LIN {X 0,Y 573.237,Z 371.706,A -85,B 0,C 180,E1 -2343.515,E2 -2343.515} C_VEL
LIN {X 0,Y 573.293,Z 371.696,A -85,B 0,C 180,E1 -2345.628,E2 -2345.628} C_VEL
LIN {X 0,Y 573.287,Z 371.699,A -85,B 0,C 180,E1 -2348.46,E2 -2348.46} C_VEL
LIN {X 0,Y 573.275,Z 371.704,A -85,B 0,C 180,E1 -2351.312,E2 -2351.312} C_VEL
LIN {X 0,Y 573.284,Z 371.701,A -85,B 0,C 180,E1 -2354.424,E2 -2354.424} C_VEL
LIN {X 0,Y 573.262,Z 371.699,A -85,B 0,C 180,E1 -2357.112,E2 -2357.112} C_VEL
LIN {X 0,Y 573.254,Z 371.701,A -85,B 0,C 180,E1 -2360.077,E2 -2360.077} C_VEL
LIN {X 0,Y 573.237,Z 371.705,A -85,B 0,C 180,E1 -2363.099,E2 -2363.099} C_VEL
LIN {X 0,Y 573.254,Z 371.702,A -85,B 0,C 180,E1 -2364.391,E2 -2364.391} C_VEL
LIN {X 0,Y 572.627,Z 371.783,A -85,B 0,C 180,E1 -2364.977,E2 -2364.977} C_VEL
LIN {X 0,Y 569.784,Z 372.141,A -85,B 0,C 180,E1 -2365.928,E2 -2365.928} C_VEL
LIN {X 0,Y 567.352,Z 372.443,A -85,B 0,C 180,E1 -2366.694,E2 -2366.694} C_VEL
LIN {X 0,Y 566.296,Z 372.571,A -85,B 0,C 180,E1 -2367.285,E2 -2367.285} C_VEL
LIN {X 0,Y 566.206,Z 372.581,A -85,B 0,C 180,E1 -2367.485,E2 -2367.485} C_VEL
LIN {X 0,Y 566.203,Z 372.58,A -85,B 0,C 180,E1 -2369.769,E2 -2369.769} C_VEL
LIN {X 0,Y 566.207,Z 372.585,A -85,B 0,C 180,E1 -2372.43,E2 -2372.43} C_VEL
LIN {X 0,Y 566.216,Z 372.578,A -85,B 0,C 180,E1 -2374.994,E2 -2374.994} C_VEL
LIN {X 0,Y 566.199,Z 372.584,A -85,B 0,C 180,E1 -2377.461,E2 -2377.461} C_VEL
LIN {X 0,Y 566.22,Z 372.579,A -85,B 0,C 180,E1 -2380.198,E2 -2380.198} C_VEL
LIN {X 0,Y 566.204,Z 372.579,A -85,B 0,C 180,E1 -2383.054,E2 -2383.054} C_VEL
LIN {X 0,Y 566.205,Z 372.58,A -85,B 0,C 180,E1 -2386.048,E2 -2386.048} C_VEL
LIN {X 0,Y 566.214,Z 372.583,A -85,B 0,C 180,E1 -2388.864,E2 -2388.864} C_VEL
LIN {X 0,Y 566.217,Z 372.582,A -85,B 0,C 180,E1 -2390.726,E2 -2390.726} C_VEL
LIN {X 0,Y 566.225,Z 373.259,A -85,B 0,C 180,E1 -2391.64,E2 -2391.64} C_VEL
LIN {X 0,Y 566.24,Z 377.975,A -85,B 0,C 180,E1 -2394.313,E2 -2394.313} C_VEL
LIN {X 0,Y 566.231,Z 382.684,A -85,B 0,C 180,E1 -2396.899,E2 -2396.899} C_VEL
LIN {X 0,Y 566.13,Z 387.389,A -85,B 0,C 180,E1 -2399.404,E2 -2399.404} C_VEL
LIN {X 0,Y 566.119,Z 392.066,A -85,B 0,C 180,E1 -2401.852,E2 -2401.852} C_VEL
LIN {X 0,Y 566.079,Z 398.311,A -85,B 0,C 180,E1 -2405.032,E2 -2405.032} C_VEL
LIN {X 0,Y 566.009,Z 403.027,A -85,B 0,C 180,E1 -2407.361,E2 -2407.361} C_VEL
LIN {X 0,Y 565.977,Z 407.753,A -85,B 0,C 180,E1 -2409.654,E2 -2409.654} C_VEL
LIN {X 0,Y 565.975,Z 412.48,A -85,B 0,C 180,E1 -2411.914,E2 -2411.914} C_VEL
LIN {X 0,Y 565.96,Z 418.537,A -85,B 0,C 180,E1 -2414.769,E2 -2414.769} C_VEL
LIN {X 0,Y 567.389,Z 426.398,A -85,B 0,C 180,E1 -2414.95,E2 -2414.95} C_VEL
LIN {X 0,Y 567.256,Z 440.824,A -85,B 0,C 180,E1 -2415.314,E2 -2415.314} C_VEL
LIN {X 0,Y 567.092,Z 455.098,A -85,B 0,C 180,E1 -2415.832,E2 -2415.832} C_VEL
LIN {X 0,Y 566.914,Z 468.271,A -85,B 0,C 180,E1 -2416.468,E2 -2416.468} C_VEL
LIN {X 0,Y 566.715,Z 480.213,A -85,B 0,C 180,E1 -2417.193,E2 -2417.193} C_VEL
LIN {X 0,Y 566.536,Z 492.291,A -85,B 0,C 180,E1 -2418.098,E2 -2418.098} C_VEL
LIN {X 0,Y 566.399,Z 503.503,A -85,B 0,C 180,E1 -2419.126,E2 -2419.126} C_VEL
LIN {X 0,Y 566.202,Z 512.969,A -85,B 0,C 180,E1 -2420.173,E2 -2420.173} C_VEL
LIN {X 0,Y 566.123,Z 521.1,A -85,B 0,C 180,E1 -2421.253,E2 -2421.253} C_VEL
LIN {X 0,Y 566.016,Z 528.883,A -85,B 0,C 180,E1 -2422.509,E2 -2422.509} C_VEL
LIN {X 0,Y 565.945,Z 534.324,A -85,B 0,C 180,E1 -2423.583,E2 -2423.583} C_VEL
LIN {X 0,Y 565.928,Z 538.8,A -85,B 0,C 180,E1 -2424.656,E2 -2424.656} C_VEL
LIN {X 0,Y 565.957,Z 542.311,A -85,B 0,C 180,E1 -2425.727,E2 -2425.727} C_VEL
LIN {X 0,Y 565.875,Z 545.743,A -85,B 0,C 180,E1 -2427.153,E2 -2427.153} C_VEL
LIN {X 0,Y 565.844,Z 547.784,A -85,B 0,C 180,E1 -2428.577,E2 -2428.577} C_VEL
LIN {X 0,Y 565.838,Z 548.496,A -85,B 0,C 180,E1 -2430,E2 -2430} C_VEL
LIN {X 0,Y 565.841,Z 547.88,A -85,B 0,C 180,E1 -2431.423,E2 -2431.423} C_VEL
LIN {X 0,Y 565.873,Z 545.922,A -85,B 0,C 180,E1 -2432.848,E2 -2432.848} C_VEL
LIN {X 0,Y 565.958,Z 542.576,A -85,B 0,C 180,E1 -2434.273,E2 -2434.273} C_VEL
LIN {X 0,Y 565.984,Z 537.747,A -85,B 0,C 180,E1 -2435.701,E2 -2435.701} C_VEL
LIN {X 0,Y 565.981,Z 531.28,A -85,B 0,C 180,E1 -2437.133,E2 -2437.133} C_VEL
LIN {X 0,Y 566.093,Z 524.08,A -85,B 0,C 180,E1 -2438.388,E2 -2438.388} C_VEL
LIN {X 0,Y 566.172,Z 516.54,A -85,B 0,C 180,E1 -2439.467,E2 -2439.467} C_VEL
LIN {X 0,Y 566.29,Z 507.484,A -85,B 0,C 180,E1 -2440.548,E2 -2440.548} C_VEL
LIN {X 0,Y 566.486,Z 498.473,A -85,B 0,C 180,E1 -2441.449,E2 -2441.449} C_VEL
LIN {X 0,Y 566.626,Z 487.721,A -85,B 0,C 180,E1 -2442.354,E2 -2442.354} C_VEL
LIN {X 0,Y 566.767,Z 475.957,A -85,B 0,C 180,E1 -2443.171,E2 -2443.171} C_VEL
LIN {X 0,Y 566.999,Z 462.98,A -85,B 0,C 180,E1 -2443.896,E2 -2443.896} C_VEL
LIN {X 0,Y 567.199,Z 450.296,A -85,B 0,C 180,E1 -2444.451,E2 -2444.451} C_VEL
LIN {X 0,Y 567.312,Z 436.696,A -85,B 0,C 180,E1 -2444.899,E2 -2444.899} C_VEL
LIN {X 0,Y 567.239,Z 424.971,A -85,B 0,C 180,E1 -2445.173,E2 -2445.173} C_VEL
LIN {X 0,Y 565.933,Z 418.532,A -85,B 0,C 180,E1 -2445.324,E2 -2445.324} C_VEL
LIN {X 0,Y 565.976,Z 412.669,A -85,B 0,C 180,E1 -2448.086,E2 -2448.086} C_VEL
LIN {X 0,Y 566.015,Z 406.364,A -85,B 0,C 180,E1 -2451.105,E2 -2451.105} C_VEL
LIN {X 0,Y 566.038,Z 400.057,A -85,B 0,C 180,E1 -2454.188,E2 -2454.188} C_VEL
LIN {X 0,Y 566.072,Z 395.207,A -85,B 0,C 180,E1 -2456.631,E2 -2456.631} C_VEL
LIN {X 0,Y 566.118,Z 390.688,A -85,B 0,C 180,E1 -2458.958,E2 -2458.958} C_VEL
LIN {X 0,Y 566.157,Z 385.986,A -85,B 0,C 180,E1 -2461.424,E2 -2461.424} C_VEL
LIN {X 0,Y 566.216,Z 381.278,A -85,B 0,C 180,E1 -2463.956,E2 -2463.956} C_VEL
LIN {X 0,Y 566.252,Z 376.566,A -85,B 0,C 180,E1 -2466.566,E2 -2466.566} C_VEL
LIN {X 0,Y 566.218,Z 373.075,A -85,B 0,C 180,E1 -2468.559,E2 -2468.559} C_VEL
LIN {X 0,Y 566.222,Z 372.584,A -85,B 0,C 180,E1 -2469.686,E2 -2469.686} C_VEL
LIN {X 0,Y 566.209,Z 372.584,A -85,B 0,C 180,E1 -2472.918,E2 -2472.918} C_VEL
LIN {X 0,Y 566.198,Z 372.584,A -85,B 0,C 180,E1 -2476.049,E2 -2476.049} C_VEL
LIN {X 0,Y 566.182,Z 372.583,A -85,B 0,C 180,E1 -2478.861,E2 -2478.861} C_VEL
LIN {X 0,Y 566.189,Z 372.582,A -85,B 0,C 180,E1 -2481.637,E2 -2481.637} C_VEL
LIN {X 0,Y 566.216,Z 372.583,A -85,B 0,C 180,E1 -2484.312,E2 -2484.312} C_VEL
LIN {X 0,Y 566.224,Z 372.577,A -85,B 0,C 180,E1 -2486.898,E2 -2486.898} C_VEL
LIN {X 0,Y 566.185,Z 372.586,A -85,B 0,C 180,E1 -2489.407,E2 -2489.407} C_VEL
LIN {X 0,Y 566.215,Z 372.578,A -85,B 0,C 180,E1 -2491.857,E2 -2491.857} C_VEL
LIN {X 0,Y 566.218,Z 372.582,A -85,B 0,C 180,E1 -2494.251,E2 -2494.251} C_VEL
LIN {X 0,Y 566.177,Z 372.582,A -85,B 0,C 180,E1 -2496.718,E2 -2496.718} C_VEL
LIN {X 0,Y 566.216,Z 372.577,A -85,B 0,C 180,E1 -2499.663,E2 -2499.663} C_VEL
LIN {X 0,Y 566.203,Z 372.58,A -85,B 0,C 180,E1 -2502.668,E2 -2502.668} C_VEL
LIN {X 0,Y 566.238,Z 372.579,A -85,B 0,C 180,E1 -2505.627,E2 -2505.627} C_VEL
LIN {X 0,Y 566.239,Z 372.581,A -85,B 0,C 180,E1 -2508.675,E2 -2508.675} C_VEL
LIN {X 0,Y 566.231,Z 372.576,A -85,B 0,C 180,E1 -2511.434,E2 -2511.434} C_VEL
LIN {X 0,Y 566.261,Z 372.572,A -85,B 0,C 180,E1 -2514.302,E2 -2514.302} C_VEL
LIN {X 0,Y 566.279,Z 372.57,A -85,B 0,C 180,E1 -2517.866,E2 -2517.866} C_VEL
LIN {X 0,Y 566.305,Z 372.566,A -85,B 0,C 180,E1 -2520.711,E2 -2520.711} C_VEL
LIN {X 0,Y 566.278,Z 372.571,A -85,B 0,C 180,E1 -2522.845,E2 -2522.845} C_VEL
LIN {X 0,Y 566.26,Z 372.572,A -85,B 0,C 180,E1 -2525.698,E2 -2525.698} C_VEL
LIN {X 0,Y 566.21,Z 372.58,A -85,B 0,C 180,E1 -2528.566,E2 -2528.566} C_VEL
LIN {X 0,Y 566.246,Z 372.579,A -85,B 0,C 180,E1 -2531.454,E2 -2531.454} C_VEL
LIN {X 0,Y 566.238,Z 372.58,A -85,B 0,C 180,E1 -2534.506,E2 -2534.506} C_VEL
LIN {X 0,Y 566.207,Z 372.579,A -85,B 0,C 180,E1 -2537.331,E2 -2537.331} C_VEL
LIN {X 0,Y 566.217,Z 372.577,A -85,B 0,C 180,E1 -2540.337,E2 -2540.337} C_VEL
LIN {X 0,Y 566.193,Z 372.58,A -85,B 0,C 180,E1 -2543.404,E2 -2543.404} C_VEL
LIN {X 0,Y 566.212,Z 372.582,A -85,B 0,C 180,E1 -2545.749,E2 -2545.749} C_VEL
LIN {X 0,Y 566.206,Z 372.579,A -85,B 0,C 180,E1 -2548.202,E2 -2548.202} C_VEL
LIN {X 0,Y 566.195,Z 372.584,A -85,B 0,C 180,E1 -2551.076,E2 -2551.076} C_VEL
LIN {X 0,Y 566.215,Z 372.58,A -85,B 0,C 180,E1 -2553.734,E2 -2553.734} C_VEL
LIN {X 0,Y 566.219,Z 372.578,A -85,B 0,C 180,E1 -2556.568,E2 -2556.568} C_VEL
LIN {X 0,Y 566.216,Z 372.578,A -85,B 0,C 180,E1 -2559.686,E2 -2559.686} C_VEL
LIN {X 0,Y 566.213,Z 372.584,A -85,B 0,C 180,E1 -2562.087,E2 -2562.087} C_VEL
LIN {X 0,Y 566.171,Z 372.585,A -85,B 0,C 180,E1 -2565.036,E2 -2565.036} C_VEL
LIN {X 0,Y 566.221,Z 372.579,A -85,B 0,C 180,E1 -2568.136,E2 -2568.136} C_VEL
LIN {X 0,Y 566.243,Z 372.603,A -85,B 0,C 180,E1 -2570.822,E2 -2570.822} C_VEL
LIN {X 0,Y 566.383,Z 376.17,A -85,B 0,C 180,E1 -2572.575,E2 -2572.575} C_VEL
LIN {X 0,Y 566.341,Z 381.706,A -85,B 0,C 180,E1 -2575.191,E2 -2575.191} C_VEL
LIN {X 0,Y 566.263,Z 387.274,A -85,B 0,C 180,E1 -2577.745,E2 -2577.745} C_VEL
LIN {X 0,Y 566.206,Z 393.116,A -85,B 0,C 180,E1 -2580.328,E2 -2580.328} C_VEL
LIN {X 0,Y 566.15,Z 400.382,A -85,B 0,C 180,E1 -2583.455,E2 -2583.455} C_VEL
LIN {X 0,Y 566.105,Z 405.984,A -85,B 0,C 180,E1 -2585.815,E2 -2585.815} C_VEL
LIN {X 0,Y 566.077,Z 413.413,A -85,B 0,C 180,E1 -2588.897,E2 -2588.897} C_VEL
LIN {X 0,Y 566.008,Z 420.842,A -85,B 0,C 180,E1 -2591.915,E2 -2591.915} C_VEL
LIN {X 0,Y 565.956,Z 427.806,A -85,B 0,C 180,E1 -2594.699,E2 -2594.699} C_VEL
LIN {X 0,Y 567.417,Z 435.018,A -85,B 0,C 180,E1 -2594.878,E2 -2594.878} C_VEL
LIN {X 0,Y 567.262,Z 449.476,A -85,B 0,C 180,E1 -2595.228,E2 -2595.228} C_VEL
LIN {X 0,Y 567.086,Z 463.96,A -85,B 0,C 180,E1 -2595.74,E2 -2595.74} C_VEL
LIN {X 0,Y 566.927,Z 477.39,A -85,B 0,C 180,E1 -2596.377,E2 -2596.377} C_VEL
LIN {X 0,Y 566.741,Z 489.51,A -85,B 0,C 180,E1 -2597.102,E2 -2597.102} C_VEL
LIN {X 0,Y 566.541,Z 501.751,A -85,B 0,C 180,E1 -2598.007,E2 -2598.007} C_VEL
LIN {X 0,Y 566.433,Z 512.501,A -85,B 0,C 180,E1 -2598.98,E2 -2598.98} C_VEL
LIN {X 0,Y 566.206,Z 521.851,A -85,B 0,C 180,E1 -2599.993,E2 -2599.993} C_VEL
LIN {X 0,Y 566.137,Z 530.172,A -85,B 0,C 180,E1 -2601.073,E2 -2601.073} C_VEL
LIN {X 0,Y 566.046,Z 538.126,A -85,B 0,C 180,E1 -2602.33,E2 -2602.33} C_VEL
LIN {X 0,Y 565.944,Z 544.527,A -85,B 0,C 180,E1 -2603.583,E2 -2603.583} C_VEL
LIN {X 0,Y 565.928,Z 548.961,A -85,B 0,C 180,E1 -2604.656,E2 -2604.656} C_VEL
LIN {X 0,Y 565.956,Z 552.443,A -85,B 0,C 180,E1 -2605.727,E2 -2605.727} C_VEL
LIN {X 0,Y 565.875,Z 555.832,A -85,B 0,C 180,E1 -2607.152,E2 -2607.152} C_VEL
LIN {X 0,Y 565.841,Z 557.833,A -85,B 0,C 180,E1 -2608.576,E2 -2608.576} C_VEL
LIN {X 0,Y 565.837,Z 558.5,A -85,B 0,C 180,E1 -2610,E2 -2610} C_VEL
LIN {X 0,Y 565.841,Z 557.833,A -85,B 0,C 180,E1 -2611.423,E2 -2611.423} C_VEL
LIN {X 0,Y 565.875,Z 555.834,A -85,B 0,C 180,E1 -2612.847,E2 -2612.847} C_VEL
LIN {X 0,Y 565.956,Z 552.445,A -85,B 0,C 180,E1 -2614.273,E2 -2614.273} C_VEL
LIN {X 0,Y 565.985,Z 547.568,A -85,B 0,C 180,E1 -2615.701,E2 -2615.701} C_VEL
LIN {X 0,Y 565.995,Z 543.045,A -85,B 0,C 180,E1 -2616.739,E2 -2616.739} C_VEL
LIN {X 0,Y 566.047,Z 536.037,A -85,B 0,C 180,E1 -2618.029,E2 -2618.029} C_VEL
LIN {X 0,Y 566.177,Z 527.559,A -85,B 0,C 180,E1 -2619.286,E2 -2619.286} C_VEL
LIN {X 0,Y 566.294,Z 518.708,A -85,B 0,C 180,E1 -2620.367,E2 -2620.367} C_VEL
LIN {X 0,Y 566.485,Z 507.99,A -85,B 0,C 180,E1 -2621.449,E2 -2621.449} C_VEL
LIN {X 0,Y 566.626,Z 497.142,A -85,B 0,C 180,E1 -2622.354,E2 -2622.354} C_VEL
LIN {X 0,Y 566.773,Z 485.258,A -85,B 0,C 180,E1 -2623.171,E2 -2623.171} C_VEL
LIN {X 0,Y 567.047,Z 472.096,A -85,B 0,C 180,E1 -2623.894,E2 -2623.894} C_VEL
LIN {X 0,Y 567.174,Z 459.298,A -85,B 0,C 180,E1 -2624.445,E2 -2624.445} C_VEL
LIN {X 0,Y 567.347,Z 445.435,A -85,B 0,C 180,E1 -2624.886,E2 -2624.886} C_VEL
LIN {X 0,Y 567.246,Z 434.169,A -85,B 0,C 180,E1 -2625.144,E2 -2625.144} C_VEL
LIN {X 0,Y 565.957,Z 427.806,A -85,B 0,C 180,E1 -2625.3,E2 -2625.3} C_VEL
LIN {X 0,Y 566.008,Z 420.842,A -85,B 0,C 180,E1 -2628.084,E2 -2628.084} C_VEL
LIN {X 0,Y 566.077,Z 413.413,A -85,B 0,C 180,E1 -2631.103,E2 -2631.103} C_VEL
LIN {X 0,Y 566.107,Z 405.985,A -85,B 0,C 180,E1 -2634.185,E2 -2634.185} C_VEL
LIN {X 0,Y 566.144,Z 400.137,A -85,B 0,C 180,E1 -2636.646,E2 -2636.646} C_VEL
LIN {X 0,Y 566.203,Z 392.884,A -85,B 0,C 180,E1 -2639.769,E2 -2639.769} C_VEL
LIN {X 0,Y 566.26,Z 386.865,A -85,B 0,C 180,E1 -2642.439,E2 -2642.439} C_VEL
LIN {X 0,Y 566.369,Z 381.254,A -85,B 0,C 180,E1 -2645.017,E2 -2645.017} C_VEL
LIN {X 0,Y 566.383,Z 376.125,A -85,B 0,C 180,E1 -2647.446,E2 -2647.446} C_VEL
LIN {X 0,Y 566.232,Z 372.582,A -85,B 0,C 180,E1 -2649.226,E2 -2649.226} C_VEL
LIN {X 0,Y 566.215,Z 372.579,A -85,B 0,C 180,E1 -2652.087,E2 -2652.087} C_VEL
LIN {X 0,Y 566.17,Z 372.586,A -85,B 0,C 180,E1 -2655.036,E2 -2655.036} C_VEL
LIN {X 0,Y 566.219,Z 372.58,A -85,B 0,C 180,E1 -2658.136,E2 -2658.136} C_VEL
LIN {X 0,Y 566.224,Z 372.579,A -85,B 0,C 180,E1 -2660.727,E2 -2660.727} C_VEL
LIN {X 0,Y 566.22,Z 372.578,A -85,B 0,C 180,E1 -2663.783,E2 -2663.783} C_VEL
LIN {X 0,Y 566.214,Z 372.581,A -85,B 0,C 180,E1 -2666.266,E2 -2666.266} C_VEL
LIN {X 0,Y 566.194,Z 372.584,A -85,B 0,C 180,E1 -2668.923,E2 -2668.923} C_VEL
LIN {X 0,Y 566.213,Z 372.578,A -85,B 0,C 180,E1 -2671.857,E2 -2671.857} C_VEL
LIN {X 0,Y 566.212,Z 372.582,A -85,B 0,C 180,E1 -2674.251,E2 -2674.251} C_VEL
LIN {X 0,Y 566.175,Z 372.583,A -85,B 0,C 180,E1 -2676.718,E2 -2676.718} C_VEL
LIN {X 0,Y 566.216,Z 372.577,A -85,B 0,C 180,E1 -2679.663,E2 -2679.663} C_VEL
LIN {X 0,Y 566.205,Z 372.58,A -85,B 0,C 180,E1 -2682.669,E2 -2682.669} C_VEL
LIN {X 0,Y 566.237,Z 372.578,A -85,B 0,C 180,E1 -2685.627,E2 -2685.627} C_VEL
LIN {X 0,Y 566.237,Z 372.581,A -85,B 0,C 180,E1 -2688.675,E2 -2688.675} C_VEL
LIN {X 0,Y 566.23,Z 372.577,A -85,B 0,C 180,E1 -2691.434,E2 -2691.434} C_VEL
LIN {X 0,Y 566.259,Z 372.572,A -85,B 0,C 180,E1 -2694.302,E2 -2694.302} C_VEL
LIN {X 0,Y 566.281,Z 372.57,A -85,B 0,C 180,E1 -2697.866,E2 -2697.866} C_VEL
LIN {X 0,Y 566.304,Z 372.567,A -85,B 0,C 180,E1 -2700.711,E2 -2700.711} C_VEL
LIN {X 0,Y 566.276,Z 372.571,A -85,B 0,C 180,E1 -2702.846,E2 -2702.846} C_VEL
LIN {X 0,Y 566.261,Z 372.572,A -85,B 0,C 180,E1 -2705.698,E2 -2705.698} C_VEL
LIN {X 0,Y 566.231,Z 372.577,A -85,B 0,C 180,E1 -2708.566,E2 -2708.566} C_VEL
LIN {X 0,Y 566.245,Z 372.579,A -85,B 0,C 180,E1 -2711.454,E2 -2711.454} C_VEL
LIN {X 0,Y 566.237,Z 372.579,A -85,B 0,C 180,E1 -2714.507,E2 -2714.507} C_VEL
LIN {X 0,Y 566.206,Z 372.579,A -85,B 0,C 180,E1 -2717.332,E2 -2717.332} C_VEL
LIN {X 0,Y 566.216,Z 372.577,A -85,B 0,C 180,E1 -2720.337,E2 -2720.337} C_VEL
LIN {X 0,Y 566.192,Z 372.581,A -85,B 0,C 180,E1 -2723.404,E2 -2723.404} C_VEL
LIN {X 0,Y 566.216,Z 372.581,A -85,B 0,C 180,E1 -2725.749,E2 -2725.749} C_VEL
LIN {X 0,Y 566.206,Z 372.581,A -85,B 0,C 180,E1 -2727.485,E2 -2727.485} C_VEL
LIN {X 0,Y 565.525,Z 372.665,A -85,B 0,C 180,E1 -2728.079,E2 -2728.079} C_VEL
LIN {X 0,Y 562.659,Z 373.025,A -85,B 0,C 180,E1 -2729.043,E2 -2729.043} C_VEL
LIN {X 0,Y 560.25,Z 373.322,A -85,B 0,C 180,E1 -2729.818,E2 -2729.818} C_VEL
LIN {X 0,Y 559.222,Z 373.45,A -85,B 0,C 180,E1 -2730.417,E2 -2730.417} C_VEL
LIN {X 0,Y 559.142,Z 373.459,A -85,B 0,C 180,E1 -2730.62,E2 -2730.62} C_VEL
LIN {X 0,Y 559.165,Z 373.457,A -85,B 0,C 180,E1 -2733.575,E2 -2733.575} C_VEL
LIN {X 0,Y 559.172,Z 373.455,A -85,B 0,C 180,E1 -2736.449,E2 -2736.449} C_VEL
LIN {X 0,Y 559.181,Z 373.46,A -85,B 0,C 180,E1 -2738.934,E2 -2738.934} C_VEL
LIN {X 0,Y 559.189,Z 373.454,A -85,B 0,C 180,E1 -2741.768,E2 -2741.768} C_VEL
LIN {X 0,Y 559.142,Z 373.459,A -85,B 0,C 180,E1 -2744.739,E2 -2744.739} C_VEL
LIN {X 0,Y 559.167,Z 373.46,A -85,B 0,C 180,E1 -2747.257,E2 -2747.257} C_VEL
LIN {X 0,Y 559.182,Z 373.459,A -85,B 0,C 180,E1 -2750.135,E2 -2750.135} C_VEL
LIN {X 0,Y 559.156,Z 373.505,A -85,B 0,C 180,E1 -2751.194,E2 -2751.194} C_VEL
LIN {X 0,Y 559.235,Z 378.005,A -85,B 0,C 180,E1 -2753.796,E2 -2753.796} C_VEL
LIN {X 0,Y 559.182,Z 382.713,A -85,B 0,C 180,E1 -2756.426,E2 -2756.426} C_VEL
LIN {X 0,Y 559.137,Z 387.415,A -85,B 0,C 180,E1 -2758.98,E2 -2758.98} C_VEL
LIN {X 0,Y 559.033,Z 393.668,A -85,B 0,C 180,E1 -2762.28,E2 -2762.28} C_VEL
LIN {X 0,Y 559.018,Z 398.653,A -85,B 0,C 180,E1 -2764.849,E2 -2764.849} C_VEL
LIN {X 0,Y 558.947,Z 404.604,A -85,B 0,C 180,E1 -2767.839,E2 -2767.839} C_VEL
LIN {X 0,Y 558.906,Z 410.906,A -85,B 0,C 180,E1 -2770.917,E2 -2770.917} C_VEL
LIN {X 0,Y 558.873,Z 415.633,A -85,B 0,C 180,E1 -2773.188,E2 -2773.188} C_VEL
LIN {X 0,Y 558.878,Z 418.705,A -85,B 0,C 180,E1 -2774.578,E2 -2774.578} C_VEL
LIN {X 0,Y 560.559,Z 427.228,A -85,B 0,C 180,E1 -2774.778,E2 -2774.778} C_VEL
LIN {X 0,Y 560.384,Z 441.221,A -85,B 0,C 180,E1 -2775.141,E2 -2775.141} C_VEL
LIN {X 0,Y 560.209,Z 455.114,A -85,B 0,C 180,E1 -2775.654,E2 -2775.654} C_VEL
LIN {X 0,Y 560,Z 468.282,A -85,B 0,C 180,E1 -2776.298,E2 -2776.298} C_VEL
LIN {X 0,Y 559.76,Z 480.22,A -85,B 0,C 180,E1 -2777.031,E2 -2777.031} C_VEL
LIN {X 0,Y 559.558,Z 492.296,A -85,B 0,C 180,E1 -2777.948,E2 -2777.948} C_VEL
LIN {X 0,Y 559.417,Z 502.3,A -85,B 0,C 180,E1 -2778.864,E2 -2778.864} C_VEL
LIN {X 0,Y 559.201,Z 511.486,A -85,B 0,C 180,E1 -2779.866,E2 -2779.866} C_VEL
LIN {X 0,Y 559.071,Z 519.868,A -85,B 0,C 180,E1 -2780.959,E2 -2780.959} C_VEL
LIN {X 0,Y 558.973,Z 527.878,A -85,B 0,C 180,E1 -2782.232,E2 -2782.232} C_VEL
LIN {X 0,Y 558.873,Z 534.327,A -85,B 0,C 180,E1 -2783.502,E2 -2783.502} C_VEL
LIN {X 0,Y 558.859,Z 538.802,A -85,B 0,C 180,E1 -2784.588,E2 -2784.588} C_VEL
LIN {X 0,Y 558.866,Z 542.314,A -85,B 0,C 180,E1 -2785.673,E2 -2785.673} C_VEL
LIN {X 0,Y 558.796,Z 545.745,A -85,B 0,C 180,E1 -2787.116,E2 -2787.116} C_VEL
LIN {X 0,Y 558.744,Z 547.785,A -85,B 0,C 180,E1 -2788.559,E2 -2788.559} C_VEL
LIN {X 0,Y 558.739,Z 548.496,A -85,B 0,C 180,E1 -2790,E2 -2790} C_VEL
LIN {X 0,Y 558.741,Z 547.879,A -85,B 0,C 180,E1 -2791.442,E2 -2791.442} C_VEL
LIN {X 0,Y 558.794,Z 545.921,A -85,B 0,C 180,E1 -2792.884,E2 -2792.884} C_VEL
LIN {X 0,Y 558.867,Z 542.575,A -85,B 0,C 180,E1 -2794.327,E2 -2794.327} C_VEL
LIN {X 0,Y 558.912,Z 537.745,A -85,B 0,C 180,E1 -2795.774,E2 -2795.774} C_VEL
LIN {X 0,Y 558.907,Z 531.278,A -85,B 0,C 180,E1 -2797.224,E2 -2797.224} C_VEL
LIN {X 0,Y 559.029,Z 524.077,A -85,B 0,C 180,E1 -2798.495,E2 -2798.495} C_VEL
LIN {X 0,Y 559.124,Z 516.536,A -85,B 0,C 180,E1 -2799.587,E2 -2799.587} C_VEL
LIN {X 0,Y 559.288,Z 507.479,A -85,B 0,C 180,E1 -2800.682,E2 -2800.682} C_VEL
LIN {X 0,Y 559.482,Z 496.513,A -85,B 0,C 180,E1 -2801.778,E2 -2801.778} C_VEL
LIN {X 0,Y 559.703,Z 485.335,A -85,B 0,C 180,E1 -2802.694,E2 -2802.694} C_VEL
LIN {X 0,Y 559.914,Z 472.981,A -85,B 0,C 180,E1 -2803.52,E2 -2803.52} C_VEL
LIN {X 0,Y 560.116,Z 461.093,A -85,B 0,C 180,E1 -2804.163,E2 -2804.163} C_VEL
LIN {X 0,Y 560.337,Z 448.009,A -85,B 0,C 180,E1 -2804.717,E2 -2804.717} C_VEL
LIN {X 0,Y 560.492,Z 434.312,A -85,B 0,C 180,E1 -2805.146,E2 -2805.146} C_VEL
LIN {X 0,Y 560.41,Z 425.983,A -85,B 0,C 180,E1 -2805.341,E2 -2805.341} C_VEL
LIN {X 0,Y 558.876,Z 418.53,A -85,B 0,C 180,E1 -2805.523,E2 -2805.523} C_VEL
LIN {X 0,Y 558.89,Z 412.668,A -85,B 0,C 180,E1 -2808.323,E2 -2808.323} C_VEL
LIN {X 0,Y 558.95,Z 406.138,A -85,B 0,C 180,E1 -2811.495,E2 -2811.495} C_VEL
LIN {X 0,Y 558.976,Z 400.098,A -85,B 0,C 180,E1 -2814.514,E2 -2814.514} C_VEL
LIN {X 0,Y 559.009,Z 395.403,A -85,B 0,C 180,E1 -2816.911,E2 -2816.911} C_VEL
LIN {X 0,Y 559.052,Z 390.721,A -85,B 0,C 180,E1 -2819.359,E2 -2819.359} C_VEL
LIN {X 0,Y 559.124,Z 386.012,A -85,B 0,C 180,E1 -2821.866,E2 -2821.866} C_VEL
LIN {X 0,Y 559.165,Z 381.307,A -85,B 0,C 180,E1 -2824.444,E2 -2824.444} C_VEL
LIN {X 0,Y 559.223,Z 376.593,A -85,B 0,C 180,E1 -2827.102,E2 -2827.102} C_VEL
LIN {X 0,Y 559.155,Z 373.463,A -85,B 0,C 180,E1 -2828.936,E2 -2828.936} C_VEL
LIN {X 0,Y 559.17,Z 373.458,A -85,B 0,C 180,E1 -2831.77,E2 -2831.77} C_VEL
LIN {X 0,Y 559.159,Z 373.459,A -85,B 0,C 180,E1 -2834.24,E2 -2834.24} C_VEL
LIN {X 0,Y 559.164,Z 373.457,A -85,B 0,C 180,E1 -2837.257,E2 -2837.257} C_VEL
LIN {X 0,Y 559.183,Z 373.454,A -85,B 0,C 180,E1 -2840.135,E2 -2840.135} C_VEL
LIN {X 0,Y 559.151,Z 373.462,A -85,B 0,C 180,E1 -2842.892,E2 -2842.892} C_VEL
LIN {X 0,Y 559.16,Z 373.458,A -85,B 0,C 180,E1 -2845.556,E2 -2845.556} C_VEL
LIN {X 0,Y 559.17,Z 373.456,A -85,B 0,C 180,E1 -2848.137,E2 -2848.137} C_VEL
LIN {X 0,Y 559.146,Z 373.462,A -85,B 0,C 180,E1 -2850.646,E2 -2850.646} C_VEL
LIN {X 0,Y 559.174,Z 373.455,A -85,B 0,C 180,E1 -2853.172,E2 -2853.172} C_VEL
LIN {X 0,Y 559.161,Z 373.46,A -85,B 0,C 180,E1 -2855.495,E2 -2855.495} C_VEL
LIN {X 0,Y 559.175,Z 373.457,A -85,B 0,C 180,E1 -2858.624,E2 -2858.624} C_VEL
LIN {X 0,Y 559.166,Z 373.458,A -85,B 0,C 180,E1 -2860.926,E2 -2860.926} C_VEL
LIN {X 0,Y 559.17,Z 373.46,A -85,B 0,C 180,E1 -2863.948,E2 -2863.948} C_VEL
LIN {X 0,Y 559.176,Z 373.454,A -85,B 0,C 180,E1 -2866.184,E2 -2866.184} C_VEL
LIN {X 0,Y 559.197,Z 373.453,A -85,B 0,C 180,E1 -2869.133,E2 -2869.133} C_VEL
LIN {X 0,Y 559.208,Z 373.455,A -85,B 0,C 180,E1 -2872.054,E2 -2872.054} C_VEL
LIN {X 0,Y 559.257,Z 373.448,A -85,B 0,C 180,E1 -2874.953,E2 -2874.953} C_VEL
LIN {X 0,Y 559.251,Z 373.446,A -85,B 0,C 180,E1 -2877.839,E2 -2877.839} C_VEL
LIN {X 0,Y 559.276,Z 373.442,A -85,B 0,C 180,E1 -2880.72,E2 -2880.72} C_VEL
LIN {X 0,Y 559.244,Z 373.448,A -85,B 0,C 180,E1 -2882.881,E2 -2882.881} C_VEL
LIN {X 0,Y 559.229,Z 373.447,A -85,B 0,C 180,E1 -2885.77,E2 -2885.77} C_VEL
LIN {X 0,Y 559.175,Z 373.455,A -85,B 0,C 180,E1 -2888.675,E2 -2888.675} C_VEL
LIN {X 0,Y 559.209,Z 373.454,A -85,B 0,C 180,E1 -2891.6,E2 -2891.6} C_VEL
LIN {X 0,Y 559.204,Z 373.457,A -85,B 0,C 180,E1 -2894.595,E2 -2894.595} C_VEL
LIN {X 0,Y 559.166,Z 373.458,A -85,B 0,C 180,E1 -2897.557,E2 -2897.557} C_VEL
LIN {X 0,Y 559.176,Z 373.457,A -85,B 0,C 180,E1 -2899.837,E2 -2899.837} C_VEL
LIN {X 0,Y 559.145,Z 373.459,A -85,B 0,C 180,E1 -2902.153,E2 -2902.153} C_VEL
LIN {X 0,Y 559.182,Z 373.454,A -85,B 0,C 180,E1 -2905.187,E2 -2905.187} C_VEL
LIN {X 0,Y 559.184,Z 373.458,A -85,B 0,C 180,E1 -2907.712,E2 -2907.712} C_VEL
LIN {X 0,Y 559.157,Z 373.456,A -85,B 0,C 180,E1 -2910.183,E2 -2910.183} C_VEL
LIN {X 0,Y 559.16,Z 373.46,A -85,B 0,C 180,E1 -2912.715,E2 -2912.715} C_VEL
LIN {X 0,Y 559.16,Z 373.459,A -85,B 0,C 180,E1 -2915.322,E2 -2915.322} C_VEL
LIN {X 0,Y 559.138,Z 373.46,A -85,B 0,C 180,E1 -2918.017,E2 -2918.017} C_VEL
LIN {X 0,Y 559.178,Z 373.458,A -85,B 0,C 180,E1 -2920.81,E2 -2920.81} C_VEL
LIN {X 0,Y 559.14,Z 373.465,A -85,B 0,C 180,E1 -2923.734,E2 -2923.734} C_VEL
LIN {X 0,Y 559.15,Z 373.462,A -85,B 0,C 180,E1 -2926.803,E2 -2926.803} C_VEL
LIN {X 0,Y 559.179,Z 373.457,A -85,B 0,C 180,E1 -2929.189,E2 -2929.189} C_VEL
LIN {X 0,Y 559.226,Z 373.554,A -85,B 0,C 180,E1 -2930.722,E2 -2930.722} C_VEL
LIN {X 0,Y 559.365,Z 376.774,A -85,B 0,C 180,E1 -2932.33,E2 -2932.33} C_VEL
LIN {X 0,Y 559.341,Z 381.817,A -85,B 0,C 180,E1 -2934.757,E2 -2934.757} C_VEL
LIN {X 0,Y 559.238,Z 387.389,A -85,B 0,C 180,E1 -2937.352,E2 -2937.352} C_VEL
LIN {X 0,Y 559.173,Z 393.578,A -85,B 0,C 180,E1 -2940.138,E2 -2940.138} C_VEL
LIN {X 0,Y 559.1,Z 400.56,A -85,B 0,C 180,E1 -2943.187,E2 -2943.187} C_VEL
LIN {X 0,Y 559.013,Z 407.827,A -85,B 0,C 180,E1 -2946.277,E2 -2946.277} C_VEL
LIN {X 0,Y 558.986,Z 415.27,A -85,B 0,C 180,E1 -2949.388,E2 -2949.388} C_VEL
LIN {X 0,Y 558.945,Z 422.699,A -85,B 0,C 180,E1 -2952.436,E2 -2952.436} C_VEL
LIN {X 0,Y 558.898,Z 427.849,A -85,B 0,C 180,E1 -2954.519,E2 -2954.519} C_VEL
LIN {X 0,Y 560.553,Z 436.545,A -85,B 0,C 180,E1 -2954.719,E2 -2954.719} C_VEL
LIN {X 0,Y 560.356,Z 450.991,A -85,B 0,C 180,E1 -2955.088,E2 -2955.088} C_VEL
LIN {X 0,Y 560.209,Z 465.083,A -85,B 0,C 180,E1 -2955.608,E2 -2955.608} C_VEL
LIN {X 0,Y 560.001,Z 477.392,A -85,B 0,C 180,E1 -2956.205,E2 -2956.205} C_VEL
LIN {X 0,Y 559.803,Z 489.512,A -85,B 0,C 180,E1 -2956.939,E2 -2956.939} C_VEL
LIN {X 0,Y 559.56,Z 501.749,A -85,B 0,C 180,E1 -2957.855,E2 -2957.855} C_VEL
LIN {X 0,Y 559.414,Z 512.773,A -85,B 0,C 180,E1 -2958.868,E2 -2958.868} C_VEL
LIN {X 0,Y 559.169,Z 523.337,A -85,B 0,C 180,E1 -2960.048,E2 -2960.048} C_VEL
LIN {X 0,Y 559.081,Z 531.407,A -85,B 0,C 180,E1 -2961.142,E2 -2961.142} C_VEL
LIN {X 0,Y 558.966,Z 539.135,A -85,B 0,C 180,E1 -2962.414,E2 -2962.414} C_VEL
LIN {X 0,Y 558.872,Z 544.527,A -85,B 0,C 180,E1 -2963.501,E2 -2963.501} C_VEL
LIN {X 0,Y 558.859,Z 548.961,A -85,B 0,C 180,E1 -2964.588,E2 -2964.588} C_VEL
LIN {X 0,Y 558.865,Z 552.443,A -85,B 0,C 180,E1 -2965.673,E2 -2965.673} C_VEL
LIN {X 0,Y 558.796,Z 555.832,A -85,B 0,C 180,E1 -2967.116,E2 -2967.116} C_VEL
LIN {X 0,Y 558.74,Z 557.833,A -85,B 0,C 180,E1 -2968.558,E2 -2968.558} C_VEL
LIN {X 0,Y 558.738,Z 558.5,A -85,B 0,C 180,E1 -2970,E2 -2970} C_VEL
LIN {X 0,Y 558.74,Z 557.834,A -85,B 0,C 180,E1 -2971.441,E2 -2971.441} C_VEL
LIN {X 0,Y 558.796,Z 555.834,A -85,B 0,C 180,E1 -2972.884,E2 -2972.884} C_VEL
LIN {X 0,Y 558.865,Z 552.445,A -85,B 0,C 180,E1 -2974.327,E2 -2974.327} C_VEL
LIN {X 0,Y 558.914,Z 547.568,A -85,B 0,C 180,E1 -2975.773,E2 -2975.773} C_VEL
LIN {X 0,Y 558.907,Z 541.054,A -85,B 0,C 180,E1 -2977.224,E2 -2977.224} C_VEL
LIN {X 0,Y 559.028,Z 533.802,A -85,B 0,C 180,E1 -2978.495,E2 -2978.495} C_VEL
LIN {X 0,Y 559.146,Z 524.823,A -85,B 0,C 180,E1 -2979.769,E2 -2979.769} C_VEL
LIN {X 0,Y 559.351,Z 515.392,A -85,B 0,C 180,E1 -2980.863,E2 -2980.863} C_VEL
LIN {X 0,Y 559.518,Z 504.952,A -85,B 0,C 180,E1 -2981.869,E2 -2981.869} C_VEL
LIN {X 0,Y 559.71,Z 493.435,A -85,B 0,C 180,E1 -2982.786,E2 -2982.786} C_VEL
LIN {X 0,Y 559.94,Z 480.643,A -85,B 0,C 180,E1 -2983.611,E2 -2983.611} C_VEL
LIN {X 0,Y 560.142,Z 468.152,A -85,B 0,C 180,E1 -2984.255,E2 -2984.255} C_VEL
LIN {X 0,Y 560.349,Z 455.044,A -85,B 0,C 180,E1 -2984.777,E2 -2984.777} C_VEL
LIN {X 0,Y 560.532,Z 440.895,A -85,B 0,C 180,E1 -2985.187,E2 -2985.187} C_VEL
LIN {X 0,Y 560.295,Z 434.755,A -85,B 0,C 180,E1 -2985.325,E2 -2985.325} C_VEL
LIN {X 0,Y 558.885,Z 427.806,A -85,B 0,C 180,E1 -2985.499,E2 -2985.499} C_VEL
LIN {X 0,Y 558.948,Z 420.842,A -85,B 0,C 180,E1 -2988.321,E2 -2988.321} C_VEL
LIN {X 0,Y 558.986,Z 415.27,A -85,B 0,C 180,E1 -2990.612,E2 -2990.612} C_VEL
LIN {X 0,Y 559.012,Z 407.811,A -85,B 0,C 180,E1 -2993.723,E2 -2993.723} C_VEL
LIN {X 0,Y 559.099,Z 400.557,A -85,B 0,C 180,E1 -2996.813,E2 -2996.813} C_VEL
LIN {X 0,Y 559.172,Z 393.57,A -85,B 0,C 180,E1 -2999.861,E2 -2999.861} C_VEL
LIN {X 0,Y 559.238,Z 387.256,A -85,B 0,C 180,E1 -3002.71,E2 -3002.71} C_VEL
LIN {X 0,Y 559.341,Z 381.68,A -85,B 0,C 180,E1 -3005.309,E2 -3005.309} C_VEL
LIN {X 0,Y 559.403,Z 376.099,A -85,B 0,C 180,E1 -3007.996,E2 -3007.996} C_VEL
LIN {X 0,Y 559.184,Z 373.46,A -85,B 0,C 180,E1 -3009.398,E2 -3009.398} C_VEL
LIN {X 0,Y 559.178,Z 373.456,A -85,B 0,C 180,E1 -3012.137,E2 -3012.137} C_VEL
LIN {X 0,Y 559.136,Z 373.461,A -85,B 0,C 180,E1 -3015.26,E2 -3015.26} C_VEL
LIN {X 0,Y 559.193,Z 373.455,A -85,B 0,C 180,E1 -3018.232,E2 -3018.232} C_VEL
LIN {X 0,Y 559.18,Z 373.459,A -85,B 0,C 180,E1 -3021.191,E2 -3021.191} C_VEL
LIN {X 0,Y 559.175,Z 373.456,A -85,B 0,C 180,E1 -3023.792,E2 -3023.792} C_VEL
LIN {X 0,Y 559.167,Z 373.457,A -85,B 0,C 180,E1 -3026.425,E2 -3026.425} C_VEL
LIN {X 0,Y 559.158,Z 373.461,A -85,B 0,C 180,E1 -3028.981,E2 -3028.981} C_VEL
LIN {X 0,Y 559.17,Z 373.455,A -85,B 0,C 180,E1 -3031.619,E2 -3031.619} C_VEL
LIN {X 0,Y 559.18,Z 373.459,A -85,B 0,C 180,E1 -3033.903,E2 -3033.903} C_VEL
LIN {X 0,Y 559.145,Z 373.458,A -85,B 0,C 180,E1 -3036.571,E2 -3036.571} C_VEL
LIN {X 0,Y 559.182,Z 373.455,A -85,B 0,C 180,E1 -3039.396,E2 -3039.396} C_VEL
LIN {X 0,Y 559.153,Z 373.458,A -85,B 0,C 180,E1 -3041.686,E2 -3041.686} C_VEL
LIN {X 0,Y 559.168,Z 373.46,A -85,B 0,C 180,E1 -3043.948,E2 -3043.948} C_VEL
LIN {X 0,Y 559.176,Z 373.454,A -85,B 0,C 180,E1 -3046.184,E2 -3046.184} C_VEL
LIN {X 0,Y 559.197,Z 373.452,A -85,B 0,C 180,E1 -3049.134,E2 -3049.134} C_VEL
LIN {X 0,Y 559.206,Z 373.454,A -85,B 0,C 180,E1 -3052.054,E2 -3052.054} C_VEL
LIN {X 0,Y 559.257,Z 373.448,A -85,B 0,C 180,E1 -3054.953,E2 -3054.953} C_VEL
LIN {X 0,Y 559.252,Z 373.445,A -85,B 0,C 180,E1 -3057.839,E2 -3057.839} C_VEL
LIN {X 0,Y 559.274,Z 373.442,A -85,B 0,C 180,E1 -3060.72,E2 -3060.72} C_VEL
LIN {X 0,Y 559.242,Z 373.448,A -85,B 0,C 180,E1 -3062.881,E2 -3062.881} C_VEL
LIN {X 0,Y 559.23,Z 373.448,A -85,B 0,C 180,E1 -3065.77,E2 -3065.77} C_VEL
LIN {X 0,Y 559.189,Z 373.453,A -85,B 0,C 180,E1 -3068.674,E2 -3068.674} C_VEL
LIN {X 0,Y 559.208,Z 373.454,A -85,B 0,C 180,E1 -3071.6,E2 -3071.6} C_VEL
LIN {X 0,Y 559.203,Z 373.457,A -85,B 0,C 180,E1 -3074.596,E2 -3074.596} C_VEL
LIN {X 0,Y 559.165,Z 373.458,A -85,B 0,C 180,E1 -3077.557,E2 -3077.557} C_VEL
LIN {X 0,Y 559.175,Z 373.457,A -85,B 0,C 180,E1 -3079.837,E2 -3079.837} C_VEL
LIN {X 0,Y 559.144,Z 373.459,A -85,B 0,C 180,E1 -3082.153,E2 -3082.153} C_VEL
LIN {X 0,Y 559.182,Z 373.454,A -85,B 0,C 180,E1 -3085.187,E2 -3085.187} C_VEL
LIN {X 0,Y 559.184,Z 373.458,A -85,B 0,C 180,E1 -3087.712,E2 -3087.712} C_VEL
LIN {X 0,Y 559.142,Z 373.459,A -85,B 0,C 180,E1 -3090.62,E2 -3090.62} C_VEL
LIN {X 0,Y 558.481,Z 373.545,A -85,B 0,C 180,E1 -3091.221,E2 -3091.221} C_VEL
LIN {X 0,Y 555.618,Z 373.901,A -85,B 0,C 180,E1 -3092.197,E2 -3092.197} C_VEL
LIN {X 0,Y 553.206,Z 374.199,A -85,B 0,C 180,E1 -3092.983,E2 -3092.983} C_VEL
LIN {X 0,Y 552.188,Z 374.326,A -85,B 0,C 180,E1 -3093.59,E2 -3093.59} C_VEL
LIN {X 0,Y 552.116,Z 374.337,A -85,B 0,C 180,E1 -3093.795,E2 -3093.795} C_VEL
LIN {X 0,Y 552.115,Z 374.335,A -85,B 0,C 180,E1 -3096.747,E2 -3096.747} C_VEL
LIN {X 0,Y 552.134,Z 374.332,A -85,B 0,C 180,E1 -3099.527,E2 -3099.527} C_VEL
LIN {X 0,Y 552.133,Z 374.336,A -85,B 0,C 180,E1 -3102.425,E2 -3102.425} C_VEL
LIN {X 0,Y 552.102,Z 374.341,A -85,B 0,C 180,E1 -3105.563,E2 -3105.563} C_VEL
LIN {X 0,Y 552.143,Z 374.337,A -85,B 0,C 180,E1 -3108.676,E2 -3108.676} C_VEL
LIN {X 0,Y 552.105,Z 374.34,A -85,B 0,C 180,E1 -3110.941,E2 -3110.941} C_VEL
LIN {X 0,Y 552.179,Z 376.458,A -85,B 0,C 180,E1 -3112.343,E2 -3112.343} C_VEL
LIN {X 0,Y 552.151,Z 381.176,A -85,B 0,C 180,E1 -3115.056,E2 -3115.056} C_VEL
LIN {X 0,Y 552.102,Z 385.883,A -85,B 0,C 180,E1 -3117.68,E2 -3117.68} C_VEL
LIN {X 0,Y 552.039,Z 390.584,A -85,B 0,C 180,E1 -3120.231,E2 -3120.231} C_VEL
LIN {X 0,Y 551.959,Z 395.875,A -85,B 0,C 180,E1 -3123.037,E2 -3123.037} C_VEL
LIN {X 0,Y 551.891,Z 401.508,A -85,B 0,C 180,E1 -3125.952,E2 -3125.952} C_VEL
LIN {X 0,Y 551.881,Z 406.294,A -85,B 0,C 180,E1 -3128.377,E2 -3128.377} C_VEL
LIN {X 0,Y 551.803,Z 412.483,A -85,B 0,C 180,E1 -3131.433,E2 -3131.433} C_VEL
LIN {X 0,Y 551.779,Z 418.392,A -85,B 0,C 180,E1 -3134.296,E2 -3134.296} C_VEL
LIN {X 0,Y 551.784,Z 418.539,A -85,B 0,C 180,E1 -3134.368,E2 -3134.368} C_VEL
LIN {X 0,Y 553.682,Z 428.899,A -85,B 0,C 180,E1 -3134.619,E2 -3134.619} C_VEL
LIN {X 0,Y 553.514,Z 442.924,A -85,B 0,C 180,E1 -3135.005,E2 -3135.005} C_VEL
LIN {X 0,Y 553.285,Z 457.197,A -85,B 0,C 180,E1 -3135.565,E2 -3135.565} C_VEL
LIN {X 0,Y 553.036,Z 469.883,A -85,B 0,C 180,E1 -3136.215,E2 -3136.215} C_VEL
LIN {X 0,Y 552.783,Z 481.521,A -85,B 0,C 180,E1 -3136.958,E2 -3136.958} C_VEL
LIN {X 0,Y 552.542,Z 493.371,A -85,B 0,C 180,E1 -3137.885,E2 -3137.885} C_VEL
LIN {X 0,Y 552.398,Z 503.77,A -85,B 0,C 180,E1 -3138.874,E2 -3138.874} C_VEL
LIN {X 0,Y 552.132,Z 512.977,A -85,B 0,C 180,E1 -3139.92,E2 -3139.92} C_VEL
LIN {X 0,Y 552.009,Z 521.107,A -85,B 0,C 180,E1 -3141.027,E2 -3141.027} C_VEL
LIN {X 0,Y 551.902,Z 528.889,A -85,B 0,C 180,E1 -3142.316,E2 -3142.316} C_VEL
LIN {X 0,Y 551.786,Z 535.436,A -85,B 0,C 180,E1 -3143.67,E2 -3143.67} C_VEL
LIN {X 0,Y 551.715,Z 540.05,A -85,B 0,C 180,E1 -3144.884,E2 -3144.884} C_VEL
LIN {X 0,Y 551.741,Z 544.21,A -85,B 0,C 180,E1 -3146.348,E2 -3146.348} C_VEL
LIN {X 0,Y 551.656,Z 546.936,A -85,B 0,C 180,E1 -3147.81,E2 -3147.81} C_VEL
LIN {X 0,Y 551.637,Z 548.306,A -85,B 0,C 180,E1 -3149.27,E2 -3149.27} C_VEL
LIN {X 0,Y 551.638,Z 548.354,A -85,B 0,C 180,E1 -3150.73,E2 -3150.73} C_VEL
LIN {X 0,Y 551.655,Z 547.069,A -85,B 0,C 180,E1 -3152.19,E2 -3152.19} C_VEL
LIN {X 0,Y 551.741,Z 544.425,A -85,B 0,C 180,E1 -3153.652,E2 -3153.652} C_VEL
LIN {X 0,Y 551.715,Z 540.352,A -85,B 0,C 180,E1 -3155.116,E2 -3155.116} C_VEL
LIN {X 0,Y 551.785,Z 535.837,A -85,B 0,C 180,E1 -3156.329,E2 -3156.329} C_VEL
LIN {X 0,Y 551.898,Z 529.381,A -85,B 0,C 180,E1 -3157.684,E2 -3157.684} C_VEL
LIN {X 0,Y 552.002,Z 521.706,A -85,B 0,C 180,E1 -3158.973,E2 -3158.973} C_VEL
LIN {X 0,Y 552.175,Z 512.213,A -85,B 0,C 180,E1 -3160.264,E2 -3160.264} C_VEL
LIN {X 0,Y 552.371,Z 501.86,A -85,B 0,C 180,E1 -3161.416,E2 -3161.416} C_VEL
LIN {X 0,Y 552.605,Z 491.19,A -85,B 0,C 180,E1 -3162.393,E2 -3162.393} C_VEL
LIN {X 0,Y 552.864,Z 478.781,A -85,B 0,C 180,E1 -3163.321,E2 -3163.321} C_VEL
LIN {X 0,Y 553.143,Z 466.484,A -85,B 0,C 180,E1 -3164.063,E2 -3164.063} C_VEL
LIN {X 0,Y 553.354,Z 452.785,A -85,B 0,C 180,E1 -3164.715,E2 -3164.715} C_VEL
LIN {X 0,Y 553.54,Z 438.632,A -85,B 0,C 180,E1 -3165.218,E2 -3165.218} C_VEL
LIN {X 0,Y 553.58,Z 427.194,A -85,B 0,C 180,E1 -3165.51,E2 -3165.51} C_VEL
LIN {X 0,Y 551.762,Z 418.529,A -85,B 0,C 180,E1 -3165.728,E2 -3165.728} C_VEL
LIN {X 0,Y 551.801,Z 414.243,A -85,B 0,C 180,E1 -3167.799,E2 -3167.799} C_VEL
LIN {X 0,Y 551.813,Z 409.514,A -85,B 0,C 180,E1 -3170.113,E2 -3170.113} C_VEL
LIN {X 0,Y 551.867,Z 404.84,A -85,B 0,C 180,E1 -3172.461,E2 -3172.461} C_VEL
LIN {X 0,Y 551.933,Z 399.258,A -85,B 0,C 180,E1 -3175.301,E2 -3175.301} C_VEL
LIN {X 0,Y 551.986,Z 393.877,A -85,B 0,C 180,E1 -3178.105,E2 -3178.105} C_VEL
LIN {X 0,Y 552.061,Z 389.182,A -85,B 0,C 180,E1 -3180.612,E2 -3180.612} C_VEL
LIN {X 0,Y 552.116,Z 384.477,A -85,B 0,C 180,E1 -3183.186,E2 -3183.186} C_VEL
LIN {X 0,Y 552.159,Z 379.763,A -85,B 0,C 180,E1 -3185.838,E2 -3185.838} C_VEL
LIN {X 0,Y 552.131,Z 375.038,A -85,B 0,C 180,E1 -3188.588,E2 -3188.588} C_VEL
LIN {X 0,Y 552.106,Z 374.341,A -85,B 0,C 180,E1 -3189.059,E2 -3189.059} C_VEL
LIN {X 0,Y 552.126,Z 374.339,A -85,B 0,C 180,E1 -3191.446,E2 -3191.446} C_VEL
LIN {X 0,Y 552.1,Z 374.342,A -85,B 0,C 180,E1 -3194.532,E2 -3194.532} C_VEL
LIN {X 0,Y 552.134,Z 374.336,A -85,B 0,C 180,E1 -3197.584,E2 -3197.584} C_VEL
LIN {X 0,Y 552.133,Z 374.332,A -85,B 0,C 180,E1 -3200.473,E2 -3200.473} C_VEL
LIN {X 0,Y 552.119,Z 374.334,A -85,B 0,C 180,E1 -3203.316,E2 -3203.316} C_VEL
LIN {X 0,Y 552.135,Z 374.337,A -85,B 0,C 180,E1 -3205.939,E2 -3205.939} C_VEL
LIN {X 0,Y 552.122,Z 374.333,A -85,B 0,C 180,E1 -3208.541,E2 -3208.541} C_VEL
LIN {X 0,Y 552.128,Z 374.333,A -85,B 0,C 180,E1 -3211.438,E2 -3211.438} C_VEL
LIN {X 0,Y 552.134,Z 374.335,A -85,B 0,C 180,E1 -3214.356,E2 -3214.356} C_VEL
LIN {X 0,Y 552.103,Z 374.335,A -85,B 0,C 180,E1 -3216.758,E2 -3216.758} C_VEL
LIN {X 0,Y 552.124,Z 374.336,A -85,B 0,C 180,E1 -3219.12,E2 -3219.12} C_VEL
LIN {X 0,Y 552.124,Z 374.333,A -85,B 0,C 180,E1 -3221.444,E2 -3221.444} C_VEL
LIN {X 0,Y 552.12,Z 374.339,A -85,B 0,C 180,E1 -3223.737,E2 -3223.737} C_VEL
LIN {X 0,Y 552.14,Z 374.331,A -85,B 0,C 180,E1 -3226.004,E2 -3226.004} C_VEL
LIN {X 0,Y 552.165,Z 374.33,A -85,B 0,C 180,E1 -3228.993,E2 -3228.993} C_VEL
LIN {X 0,Y 552.162,Z 374.335,A -85,B 0,C 180,E1 -3231.952,E2 -3231.952} C_VEL
LIN {X 0,Y 552.232,Z 374.322,A -85,B 0,C 180,E1 -3234.889,E2 -3234.889} C_VEL
LIN {X 0,Y 552.223,Z 374.321,A -85,B 0,C 180,E1 -3237.812,E2 -3237.812} C_VEL
LIN {X 0,Y 552.246,Z 374.317,A -85,B 0,C 180,E1 -3240.729,E2 -3240.729} C_VEL
LIN {X 0,Y 552.211,Z 374.324,A -85,B 0,C 180,E1 -3242.918,E2 -3242.918} C_VEL
LIN {X 0,Y 552.2,Z 374.323,A -85,B 0,C 180,E1 -3245.844,E2 -3245.844} C_VEL
LIN {X 0,Y 552.15,Z 374.33,A -85,B 0,C 180,E1 -3248.786,E2 -3248.786} C_VEL
LIN {X 0,Y 552.167,Z 374.329,A -85,B 0,C 180,E1 -3251.75,E2 -3251.75} C_VEL
LIN {X 0,Y 552.14,Z 374.336,A -85,B 0,C 180,E1 -3254.748,E2 -3254.748} C_VEL
LIN {X 0,Y 552.117,Z 374.339,A -85,B 0,C 180,E1 -3257.788,E2 -3257.788} C_VEL
LIN {X 0,Y 552.134,Z 374.332,A -85,B 0,C 180,E1 -3260.101,E2 -3260.101} C_VEL
LIN {X 0,Y 552.099,Z 374.339,A -85,B 0,C 180,E1 -3262.451,E2 -3262.451} C_VEL
LIN {X 0,Y 552.158,Z 374.329,A -85,B 0,C 180,E1 -3265.35,E2 -3265.35} C_VEL
LIN {X 0,Y 552.123,Z 374.334,A -85,B 0,C 180,E1 -3268.098,E2 -3268.098} C_VEL
LIN {X 0,Y 552.106,Z 374.338,A -85,B 0,C 180,E1 -3270.609,E2 -3270.609} C_VEL
LIN {X 0,Y 552.119,Z 374.334,A -85,B 0,C 180,E1 -3273.186,E2 -3273.186} C_VEL
LIN {X 0,Y 552.116,Z 374.339,A -85,B 0,C 180,E1 -3275.841,E2 -3275.841} C_VEL
LIN {X 0,Y 552.129,Z 374.338,A -85,B 0,C 180,E1 -3279.062,E2 -3279.062} C_VEL
LIN {X 0,Y 552.14,Z 374.332,A -85,B 0,C 180,E1 -3281.444,E2 -3281.444} C_VEL
LIN {X 0,Y 552.093,Z 374.337,A -85,B 0,C 180,E1 -3284.531,E2 -3284.531} C_VEL
LIN {X 0,Y 552.134,Z 374.335,A -85,B 0,C 180,E1 -3287.584,E2 -3287.584} C_VEL
LIN {X 0,Y 552.173,Z 374.501,A -85,B 0,C 180,E1 -3290.614,E2 -3290.614} C_VEL
LIN {X 0,Y 552.346,Z 377.936,A -85,B 0,C 180,E1 -3292.356,E2 -3292.356} C_VEL
LIN {X 0,Y 552.28,Z 383.512,A -85,B 0,C 180,E1 -3295.065,E2 -3295.065} C_VEL
LIN {X 0,Y 552.201,Z 389.096,A -85,B 0,C 180,E1 -3297.687,E2 -3297.687} C_VEL
LIN {X 0,Y 552.129,Z 394.691,A -85,B 0,C 180,E1 -3300.236,E2 -3300.236} C_VEL
LIN {X 0,Y 552.052,Z 400.982,A -85,B 0,C 180,E1 -3303.018,E2 -3303.018} C_VEL
LIN {X 0,Y 551.968,Z 407.793,A -85,B 0,C 180,E1 -3305.956,E2 -3305.956} C_VEL
LIN {X 0,Y 551.947,Z 413.475,A -85,B 0,C 180,E1 -3308.36,E2 -3308.36} C_VEL
LIN {X 0,Y 551.891,Z 418.984,A -85,B 0,C 180,E1 -3310.665,E2 -3310.665} C_VEL
LIN {X 0,Y 551.862,Z 424.556,A -85,B 0,C 180,E1 -3312.968,E2 -3312.968} C_VEL
LIN {X 0,Y 551.794,Z 427.849,A -85,B 0,C 180,E1 -3314.314,E2 -3314.314} C_VEL
LIN {X 0,Y 553.721,Z 438.057,A -85,B 0,C 180,E1 -3314.557,E2 -3314.557} C_VEL
LIN {X 0,Y 553.504,Z 452.273,A -85,B 0,C 180,E1 -3314.939,E2 -3314.939} C_VEL
LIN {X 0,Y 553.302,Z 466.163,A -85,B 0,C 180,E1 -3315.471,E2 -3315.471} C_VEL
LIN {X 0,Y 553.074,Z 479.056,A -85,B 0,C 180,E1 -3316.122,E2 -3316.122} C_VEL
LIN {X 0,Y 552.784,Z 492.139,A -85,B 0,C 180,E1 -3316.958,E2 -3316.958} C_VEL
LIN {X 0,Y 552.534,Z 503.886,A -85,B 0,C 180,E1 -3317.885,E2 -3317.885} C_VEL
LIN {X 0,Y 552.395,Z 514.223,A -85,B 0,C 180,E1 -3318.876,E2 -3318.876} C_VEL
LIN {X 0,Y 552.121,Z 523.337,A -85,B 0,C 180,E1 -3319.92,E2 -3319.92} C_VEL
LIN {X 0,Y 552.011,Z 531.406,A -85,B 0,C 180,E1 -3321.027,E2 -3321.027} C_VEL
LIN {X 0,Y 551.901,Z 539.134,A -85,B 0,C 180,E1 -3322.316,E2 -3322.316} C_VEL
LIN {X 0,Y 551.785,Z 545.634,A -85,B 0,C 180,E1 -3323.669,E2 -3323.669} C_VEL
LIN {X 0,Y 551.716,Z 550.2,A -85,B 0,C 180,E1 -3324.884,E2 -3324.884} C_VEL
LIN {X 0,Y 551.74,Z 554.316,A -85,B 0,C 180,E1 -3326.348,E2 -3326.348} C_VEL
LIN {X 0,Y 551.656,Z 557.001,A -85,B 0,C 180,E1 -3327.81,E2 -3327.81} C_VEL
LIN {X 0,Y 551.639,Z 558.333,A -85,B 0,C 180,E1 -3329.27,E2 -3329.27} C_VEL
LIN {X 0,Y 551.639,Z 558.333,A -85,B 0,C 180,E1 -3330.73,E2 -3330.73} C_VEL
LIN {X 0,Y 551.656,Z 557.003,A -85,B 0,C 180,E1 -3332.19,E2 -3332.19} C_VEL
LIN {X 0,Y 551.74,Z 554.319,A -85,B 0,C 180,E1 -3333.652,E2 -3333.652} C_VEL
LIN {X 0,Y 551.716,Z 550.202,A -85,B 0,C 180,E1 -3335.116,E2 -3335.116} C_VEL
LIN {X 0,Y 551.798,Z 545.574,A -85,B 0,C 180,E1 -3336.344,E2 -3336.344} C_VEL
LIN {X 0,Y 551.901,Z 539.135,A -85,B 0,C 180,E1 -3337.684,E2 -3337.684} C_VEL
LIN {X 0,Y 552.011,Z 531.407,A -85,B 0,C 180,E1 -3338.973,E2 -3338.973} C_VEL
LIN {X 0,Y 552.121,Z 523.338,A -85,B 0,C 180,E1 -3340.08,E2 -3340.08} C_VEL
LIN {X 0,Y 552.401,Z 513.09,A -85,B 0,C 180,E1 -3341.242,E2 -3341.242} C_VEL
LIN {X 0,Y 552.592,Z 501.749,A -85,B 0,C 180,E1 -3342.3,E2 -3342.3} C_VEL
LIN {X 0,Y 552.861,Z 489.518,A -85,B 0,C 180,E1 -3343.227,E2 -3343.227} C_VEL
LIN {X 0,Y 553.098,Z 477.399,A -85,B 0,C 180,E1 -3343.971,E2 -3343.971} C_VEL
LIN {X 0,Y 553.291,Z 463.959,A -85,B 0,C 180,E1 -3344.623,E2 -3344.623} C_VEL
LIN {X 0,Y 553.56,Z 449.679,A -85,B 0,C 180,E1 -3345.14,E2 -3345.14} C_VEL
LIN {X 0,Y 553.55,Z 436.293,A -85,B 0,C 180,E1 -3345.484,E2 -3345.484} C_VEL
LIN {X 0,Y 551.8,Z 427.806,A -85,B 0,C 180,E1 -3345.703,E2 -3345.703} C_VEL
LIN {X 0,Y 551.86,Z 422.699,A -85,B 0,C 180,E1 -3347.797,E2 -3347.797} C_VEL
LIN {X 0,Y 551.917,Z 417.128,A -85,B 0,C 180,E1 -3350.109,E2 -3350.109} C_VEL
LIN {X 0,Y 551.937,Z 411.509,A -85,B 0,C 180,E1 -3352.458,E2 -3352.458} C_VEL
LIN {X 0,Y 551.998,Z 404.812,A -85,B 0,C 180,E1 -3355.315,E2 -3355.315} C_VEL
LIN {X 0,Y 552.047,Z 398.432,A -85,B 0,C 180,E1 -3358.102,E2 -3358.102} C_VEL
LIN {X 0,Y 552.117,Z 392.815,A -85,B 0,C 180,E1 -3360.608,E2 -3360.608} C_VEL
LIN {X 0,Y 552.22,Z 387.233,A -85,B 0,C 180,E1 -3363.179,E2 -3363.179} C_VEL
LIN {X 0,Y 552.319,Z 381.651,A -85,B 0,C 180,E1 -3365.826,E2 -3365.826} C_VEL
LIN {X 0,Y 552.356,Z 376.081,A -85,B 0,C 180,E1 -3368.569,E2 -3368.569} C_VEL
LIN {X 0,Y 552.163,Z 374.335,A -85,B 0,C 180,E1 -3369.524,E2 -3369.524} C_VEL
LIN {X 0,Y 552.132,Z 374.335,A -85,B 0,C 180,E1 -3372.425,E2 -3372.425} C_VEL
LIN {X 0,Y 552.095,Z 374.338,A -85,B 0,C 180,E1 -3375.562,E2 -3375.562} C_VEL
LIN {X 0,Y 552.142,Z 374.332,A -85,B 0,C 180,E1 -3378.676,E2 -3378.676} C_VEL
LIN {X 0,Y 552.122,Z 374.336,A -85,B 0,C 180,E1 -3381.411,E2 -3381.411} C_VEL
LIN {X 0,Y 552.115,Z 374.339,A -85,B 0,C 180,E1 -3384.159,E2 -3384.159} C_VEL
LIN {X 0,Y 552.125,Z 374.333,A -85,B 0,C 180,E1 -3386.815,E2 -3386.815} C_VEL
LIN {X 0,Y 552.105,Z 374.34,A -85,B 0,C 180,E1 -3389.391,E2 -3389.391} C_VEL
LIN {X 0,Y 552.121,Z 374.334,A -85,B 0,C 180,E1 -3391.902,E2 -3391.902} C_VEL
LIN {X 0,Y 552.157,Z 374.329,A -85,B 0,C 180,E1 -3394.65,E2 -3394.65} C_VEL
LIN {X 0,Y 552.095,Z 374.34,A -85,B 0,C 180,E1 -3397.549,E2 -3397.549} C_VEL
LIN {X 0,Y 552.151,Z 374.334,A -85,B 0,C 180,E1 -3400.374,E2 -3400.374} C_VEL
LIN {X 0,Y 552.158,Z 374.328,A -85,B 0,C 180,E1 -3402.977,E2 -3402.977} C_VEL
LIN {X 0,Y 552.139,Z 374.331,A -85,B 0,C 180,E1 -3406.005,E2 -3406.005} C_VEL
LIN {X 0,Y 552.165,Z 374.329,A -85,B 0,C 180,E1 -3408.993,E2 -3408.993} C_VEL
LIN {X 0,Y 552.16,Z 374.333,A -85,B 0,C 180,E1 -3411.952,E2 -3411.952} C_VEL
LIN {X 0,Y 552.232,Z 374.323,A -85,B 0,C 180,E1 -3414.889,E2 -3414.889} C_VEL
LIN {X 0,Y 552.224,Z 374.321,A -85,B 0,C 180,E1 -3417.812,E2 -3417.812} C_VEL
LIN {X 0,Y 552.245,Z 374.318,A -85,B 0,C 180,E1 -3420.729,E2 -3420.729} C_VEL
LIN {X 0,Y 552.209,Z 374.324,A -85,B 0,C 180,E1 -3422.918,E2 -3422.918} C_VEL
LIN {X 0,Y 552.201,Z 374.324,A -85,B 0,C 180,E1 -3425.844,E2 -3425.844} C_VEL
LIN {X 0,Y 552.16,Z 374.328,A -85,B 0,C 180,E1 -3428.786,E2 -3428.786} C_VEL
LIN {X 0,Y 552.165,Z 374.33,A -85,B 0,C 180,E1 -3431.751,E2 -3431.751} C_VEL
LIN {X 0,Y 552.139,Z 374.336,A -85,B 0,C 180,E1 -3434.748,E2 -3434.748} C_VEL
LIN {X 0,Y 552.116,Z 374.339,A -85,B 0,C 180,E1 -3437.788,E2 -3437.788} C_VEL
LIN {X 0,Y 552.133,Z 374.332,A -85,B 0,C 180,E1 -3440.101,E2 -3440.101} C_VEL
LIN {X 0,Y 552.099,Z 374.339,A -85,B 0,C 180,E1 -3442.451,E2 -3442.451} C_VEL
LIN {X 0,Y 552.158,Z 374.329,A -85,B 0,C 180,E1 -3445.35,E2 -3445.35} C_VEL
LIN {X 0,Y 552.122,Z 374.334,A -85,B 0,C 180,E1 -3448.098,E2 -3448.098} C_VEL
LIN {X 0,Y 552.105,Z 374.339,A -85,B 0,C 180,E1 -3450.616,E2 -3450.616} C_VEL
LIN {X 0,Y 552.118,Z 374.334,A -85,B 0,C 180,E1 -3453.186,E2 -3453.186} C_VEL
LIN {X 0,Y 552.116,Z 374.337,A -85,B 0,C 180,E1 -3453.795,E2 -3453.795} C_VEL
LIN {X 0,Y 551.477,Z 374.42,A -85,B 0,C 180,E1 -3454.404,E2 -3454.404} C_VEL
LIN {X 0,Y 548.635,Z 374.771,A -85,B 0,C 180,E1 -3455.392,E2 -3455.392} C_VEL
LIN {X 0,Y 546.211,Z 375.071,A -85,B 0,C 180,E1 -3456.187,E2 -3456.187} C_VEL
LIN {X 0,Y 545.163,Z 375.201,A -85,B 0,C 180,E1 -3456.801,E2 -3456.801} C_VEL
LIN {X 0,Y 545.074,Z 375.214,A -85,B 0,C 180,E1 -3457.009,E2 -3457.009} C_VEL
LIN {X 0,Y 545.074,Z 375.213,A -85,B 0,C 180,E1 -3460.142,E2 -3460.142} C_VEL
LIN {X 0,Y 545.081,Z 375.211,A -85,B 0,C 180,E1 -3463.107,E2 -3463.107} C_VEL
LIN {X 0,Y 545.068,Z 375.213,A -85,B 0,C 180,E1 -3466.224,E2 -3466.224} C_VEL
LIN {X 0,Y 545.1,Z 375.213,A -85,B 0,C 180,E1 -3468.887,E2 -3468.887} C_VEL
LIN {X 0,Y 545.064,Z 375.218,A -85,B 0,C 180,E1 -3470.817,E2 -3470.817} C_VEL
LIN {X 0,Y 545.143,Z 378.061,A -85,B 0,C 180,E1 -3472.705,E2 -3472.705} C_VEL
LIN {X 0,Y 545.132,Z 383.055,A -85,B 0,C 180,E1 -3475.599,E2 -3475.599} C_VEL
LIN {X 0,Y 545.044,Z 387.918,A -85,B 0,C 180,E1 -3478.324,E2 -3478.324} C_VEL
LIN {X 0,Y 544.963,Z 393.759,A -85,B 0,C 180,E1 -3481.5,E2 -3481.5} C_VEL
LIN {X 0,Y 544.887,Z 399.983,A -85,B 0,C 180,E1 -3484.809,E2 -3484.809} C_VEL
LIN {X 0,Y 544.81,Z 406.23,A -85,B 0,C 180,E1 -3488.031,E2 -3488.031} C_VEL
LIN {X 0,Y 544.763,Z 410.921,A -85,B 0,C 180,E1 -3490.402,E2 -3490.402} C_VEL
LIN {X 0,Y 544.683,Z 417.211,A -85,B 0,C 180,E1 -3493.509,E2 -3493.509} C_VEL
LIN {X 0,Y 544.697,Z 418.681,A -85,B 0,C 180,E1 -3494.165,E2 -3494.165} C_VEL
LIN {X 0,Y 546.825,Z 429.527,A -85,B 0,C 180,E1 -3494.434,E2 -3494.434} C_VEL
LIN {X 0,Y 546.656,Z 443.786,A -85,B 0,C 180,E1 -3494.843,E2 -3494.843} C_VEL
LIN {X 0,Y 546.422,Z 457.208,A -85,B 0,C 180,E1 -3495.38,E2 -3495.38} C_VEL
LIN {X 0,Y 546.126,Z 469.891,A -85,B 0,C 180,E1 -3496.037,E2 -3496.037} C_VEL
LIN {X 0,Y 545.82,Z 482.817,A -85,B 0,C 180,E1 -3496.883,E2 -3496.883} C_VEL
LIN {X 0,Y 545.552,Z 494.445,A -85,B 0,C 180,E1 -3497.822,E2 -3497.822} C_VEL
LIN {X 0,Y 545.339,Z 504.968,A -85,B 0,C 180,E1 -3498.854,E2 -3498.854} C_VEL
LIN {X 0,Y 545.091,Z 514.467,A -85,B 0,C 180,E1 -3499.976,E2 -3499.976} C_VEL
LIN {X 0,Y 544.911,Z 523.533,A -85,B 0,C 180,E1 -3501.284,E2 -3501.284} C_VEL
LIN {X 0,Y 544.784,Z 530.835,A -85,B 0,C 180,E1 -3502.588,E2 -3502.588} C_VEL
LIN {X 0,Y 544.732,Z 537.396,A -85,B 0,C 180,E1 -3504.076,E2 -3504.076} C_VEL
LIN {X 0,Y 544.654,Z 542.318,A -85,B 0,C 180,E1 -3505.56,E2 -3505.56} C_VEL
LIN {X 0,Y 544.647,Z 545.748,A -85,B 0,C 180,E1 -3507.041,E2 -3507.041} C_VEL
LIN {X 0,Y 544.544,Z 547.788,A -85,B 0,C 180,E1 -3508.521,E2 -3508.521} C_VEL
LIN {X 0,Y 544.54,Z 548.496,A -85,B 0,C 180,E1 -3510,E2 -3510} C_VEL
LIN {X 0,Y 544.542,Z 547.878,A -85,B 0,C 180,E1 -3511.479,E2 -3511.479} C_VEL
LIN {X 0,Y 544.646,Z 545.919,A -85,B 0,C 180,E1 -3512.959,E2 -3512.959} C_VEL
LIN {X 0,Y 544.655,Z 542.572,A -85,B 0,C 180,E1 -3514.44,E2 -3514.44} C_VEL
LIN {X 0,Y 544.73,Z 537.741,A -85,B 0,C 180,E1 -3515.924,E2 -3515.924} C_VEL
LIN {X 0,Y 544.784,Z 531.273,A -85,B 0,C 180,E1 -3517.412,E2 -3517.412} C_VEL
LIN {X 0,Y 544.906,Z 524.071,A -85,B 0,C 180,E1 -3518.717,E2 -3518.717} C_VEL
LIN {X 0,Y 545.04,Z 516.528,A -85,B 0,C 180,E1 -3519.837,E2 -3519.837} C_VEL
LIN {X 0,Y 545.276,Z 507.468,A -85,B 0,C 180,E1 -3520.959,E2 -3520.959} C_VEL
LIN {X 0,Y 545.506,Z 496.499,A -85,B 0,C 180,E1 -3522.085,E2 -3522.085} C_VEL
LIN {X 0,Y 545.786,Z 485.321,A -85,B 0,C 180,E1 -3523.023,E2 -3523.023} C_VEL
LIN {X 0,Y 546.064,Z 472.964,A -85,B 0,C 180,E1 -3523.869,E2 -3523.869} C_VEL
LIN {X 0,Y 546.335,Z 461.072,A -85,B 0,C 180,E1 -3524.528,E2 -3524.528} C_VEL
LIN {X 0,Y 546.591,Z 449.032,A -85,B 0,C 180,E1 -3525.057,E2 -3525.057} C_VEL
LIN {X 0,Y 546.732,Z 435.865,A -85,B 0,C 180,E1 -3525.495,E2 -3525.495} C_VEL
LIN {X 0,Y 546.707,Z 428.186,A -85,B 0,C 180,E1 -3525.688,E2 -3525.688} C_VEL
LIN {X 0,Y 544.694,Z 418.528,A -85,B 0,C 180,E1 -3525.937,E2 -3525.937} C_VEL
LIN {X 0,Y 544.729,Z 412.667,A -85,B 0,C 180,E1 -3528.817,E2 -3528.817} C_VEL
LIN {X 0,Y 544.811,Z 406.461,A -85,B 0,C 180,E1 -3531.969,E2 -3531.969} C_VEL
LIN {X 0,Y 544.888,Z 400.186,A -85,B 0,C 180,E1 -3535.191,E2 -3535.191} C_VEL
LIN {X 0,Y 544.964,Z 393.911,A -85,B 0,C 180,E1 -3538.5,E2 -3538.5} C_VEL
LIN {X 0,Y 545.045,Z 388.08,A -85,B 0,C 180,E1 -3541.676,E2 -3541.676} C_VEL
LIN {X 0,Y 545.091,Z 382.935,A -85,B 0,C 180,E1 -3544.563,E2 -3544.563} C_VEL
LIN {X 0,Y 545.151,Z 378.215,A -85,B 0,C 180,E1 -3547.295,E2 -3547.295} C_VEL
LIN {X 0,Y 545.065,Z 375.218,A -85,B 0,C 180,E1 -3549.183,E2 -3549.183} C_VEL
LIN {X 0,Y 545.081,Z 375.212,A -85,B 0,C 180,E1 -3552.103,E2 -3552.103} C_VEL
LIN {X 0,Y 545.065,Z 375.214,A -85,B 0,C 180,E1 -3555.167,E2 -3555.167} C_VEL
LIN {X 0,Y 545.084,Z 375.217,A -85,B 0,C 180,E1 -3557.897,E2 -3557.897} C_VEL
LIN {X 0,Y 545.084,Z 375.213,A -85,B 0,C 180,E1 -3560.818,E2 -3560.818} C_VEL
LIN {X 0,Y 545.06,Z 375.213,A -85,B 0,C 180,E1 -3563.621,E2 -3563.621} C_VEL
LIN {X 0,Y 545.072,Z 375.214,A -85,B 0,C 180,E1 -3566.328,E2 -3566.328} C_VEL
LIN {X 0,Y 545.07,Z 375.214,A -85,B 0,C 180,E1 -3568.952,E2 -3568.952} C_VEL
LIN {X 0,Y 545.106,Z 375.208,A -85,B 0,C 180,E1 -3571.508,E2 -3571.508} C_VEL
LIN {X 0,Y 545.099,Z 375.21,A -85,B 0,C 180,E1 -3574.491,E2 -3574.491} C_VEL
LIN {X 0,Y 545.042,Z 375.22,A -85,B 0,C 180,E1 -3577.242,E2 -3577.242} C_VEL
LIN {X 0,Y 545.121,Z 375.208,A -85,B 0,C 180,E1 -3580.415,E2 -3580.415} C_VEL
LIN {X 0,Y 545.076,Z 375.213,A -85,B 0,C 180,E1 -3583.521,E2 -3583.521} C_VEL
LIN {X 0,Y 545.099,Z 375.21,A -85,B 0,C 180,E1 -3585.82,E2 -3585.82} C_VEL
LIN {X 0,Y 545.121,Z 375.21,A -85,B 0,C 180,E1 -3588.849,E2 -3588.849} C_VEL
LIN {X 0,Y 545.132,Z 375.209,A -85,B 0,C 180,E1 -3591.847,E2 -3591.847} C_VEL
LIN {X 0,Y 545.207,Z 375.197,A -85,B 0,C 180,E1 -3594.823,E2 -3594.823} C_VEL
LIN {X 0,Y 545.196,Z 375.196,A -85,B 0,C 180,E1 -3597.784,E2 -3597.784} C_VEL
LIN {X 0,Y 545.216,Z 375.193,A -85,B 0,C 180,E1 -3600.739,E2 -3600.739} C_VEL
LIN {X 0,Y 545.177,Z 375.201,A -85,B 0,C 180,E1 -3602.956,E2 -3602.956} C_VEL
LIN {X 0,Y 545.172,Z 375.199,A -85,B 0,C 180,E1 -3605.919,E2 -3605.919} C_VEL
LIN {X 0,Y 545.112,Z 375.206,A -85,B 0,C 180,E1 -3608.9,E2 -3608.9} C_VEL
LIN {X 0,Y 545.139,Z 375.204,A -85,B 0,C 180,E1 -3611.904,E2 -3611.904} C_VEL
LIN {X 0,Y 545.089,Z 375.212,A -85,B 0,C 180,E1 -3614.943,E2 -3614.943} C_VEL
LIN {X 0,Y 545.085,Z 375.214,A -85,B 0,C 180,E1 -3618.026,E2 -3618.026} C_VEL
LIN {X 0,Y 545.099,Z 375.208,A -85,B 0,C 180,E1 -3620.372,E2 -3620.372} C_VEL
LIN {X 0,Y 545.095,Z 375.208,A -85,B 0,C 180,E1 -3623.559,E2 -3623.559} C_VEL
LIN {X 0,Y 545.081,Z 375.216,A -85,B 0,C 180,E1 -3626,E2 -3626} C_VEL
LIN {X 0,Y 545.092,Z 375.21,A -85,B 0,C 180,E1 -3628.748,E2 -3628.748} C_VEL
LIN {X 0,Y 545.06,Z 375.213,A -85,B 0,C 180,E1 -3631.679,E2 -3631.679} C_VEL
LIN {X 0,Y 545.084,Z 375.211,A -85,B 0,C 180,E1 -3634.563,E2 -3634.563} C_VEL
LIN {X 0,Y 545.043,Z 375.222,A -85,B 0,C 180,E1 -3637.303,E2 -3637.303} C_VEL
LIN {X 0,Y 545.095,Z 375.211,A -85,B 0,C 180,E1 -3640.14,E2 -3640.14} C_VEL
LIN {X 0,Y 545.081,Z 375.211,A -85,B 0,C 180,E1 -3643.106,E2 -3643.106} C_VEL
LIN {X 0,Y 545.069,Z 375.213,A -85,B 0,C 180,E1 -3646.224,E2 -3646.224} C_VEL
LIN {X 0,Y 545.1,Z 375.214,A -85,B 0,C 180,E1 -3648.887,E2 -3648.887} C_VEL
LIN {X 0,Y 545.119,Z 375.253,A -85,B 0,C 180,E1 -3650.403,E2 -3650.403} C_VEL
LIN {X 0,Y 545.374,Z 377.976,A -85,B 0,C 180,E1 -3651.821,E2 -3651.821} C_VEL
LIN {X 0,Y 545.288,Z 383.485,A -85,B 0,C 180,E1 -3654.55,E2 -3654.55} C_VEL
LIN {X 0,Y 545.175,Z 389.065,A -85,B 0,C 180,E1 -3657.219,E2 -3657.219} C_VEL
LIN {X 0,Y 545.105,Z 394.653,A -85,B 0,C 180,E1 -3659.813,E2 -3659.813} C_VEL
LIN {X 0,Y 544.988,Z 401.418,A -85,B 0,C 180,E1 -3662.849,E2 -3662.849} C_VEL
LIN {X 0,Y 544.914,Z 407.759,A -85,B 0,C 180,E1 -3665.624,E2 -3665.624} C_VEL
LIN {X 0,Y 544.893,Z 413.818,A -85,B 0,C 180,E1 -3668.226,E2 -3668.226} C_VEL
LIN {X 0,Y 544.787,Z 420.842,A -85,B 0,C 180,E1 -3671.185,E2 -3671.185} C_VEL
LIN {X 0,Y 544.751,Z 427.849,A -85,B 0,C 180,E1 -3674.106,E2 -3674.106} C_VEL
LIN {X 0,Y 546.869,Z 438.899,A -85,B 0,C 180,E1 -3674.376,E2 -3674.376} C_VEL
LIN {X 0,Y 546.641,Z 453,A -85,B 0,C 180,E1 -3674.769,E2 -3674.769} C_VEL
LIN {X 0,Y 546.397,Z 466.162,A -85,B 0,C 180,E1 -3675.284,E2 -3675.284} C_VEL
LIN {X 0,Y 546.153,Z 479.054,A -85,B 0,C 180,E1 -3675.943,E2 -3675.943} C_VEL
LIN {X 0,Y 545.857,Z 492.137,A -85,B 0,C 180,E1 -3676.789,E2 -3676.789} C_VEL
LIN {X 0,Y 545.543,Z 503.885,A -85,B 0,C 180,E1 -3677.727,E2 -3677.727} C_VEL
LIN {X 0,Y 545.389,Z 513.677,A -85,B 0,C 180,E1 -3678.674,E2 -3678.674} C_VEL
LIN {X 0,Y 545.101,Z 523.337,A -85,B 0,C 180,E1 -3679.789,E2 -3679.789} C_VEL
LIN {X 0,Y 544.969,Z 531.405,A -85,B 0,C 180,E1 -3680.91,E2 -3680.91} C_VEL
LIN {X 0,Y 544.824,Z 539.134,A -85,B 0,C 180,E1 -3682.216,E2 -3682.216} C_VEL
LIN {X 0,Y 544.753,Z 544.875,A -85,B 0,C 180,E1 -3683.412,E2 -3683.412} C_VEL
LIN {X 0,Y 544.646,Z 550.201,A -85,B 0,C 180,E1 -3684.818,E2 -3684.818} C_VEL
LIN {X 0,Y 544.657,Z 554.316,A -85,B 0,C 180,E1 -3686.301,E2 -3686.301} C_VEL
LIN {X 0,Y 544.57,Z 557.002,A -85,B 0,C 180,E1 -3687.781,E2 -3687.781} C_VEL
LIN {X 0,Y 544.539,Z 558.333,A -85,B 0,C 180,E1 -3689.26,E2 -3689.26} C_VEL
LIN {X 0,Y 544.539,Z 558.334,A -85,B 0,C 180,E1 -3690.739,E2 -3690.739} C_VEL
LIN {X 0,Y 544.57,Z 557.004,A -85,B 0,C 180,E1 -3692.219,E2 -3692.219} C_VEL
LIN {X 0,Y 544.657,Z 554.32,A -85,B 0,C 180,E1 -3693.699,E2 -3693.699} C_VEL
LIN {X 0,Y 544.646,Z 550.202,A -85,B 0,C 180,E1 -3695.182,E2 -3695.182} C_VEL
LIN {X 0,Y 544.738,Z 544.936,A -85,B 0,C 180,E1 -3696.573,E2 -3696.573} C_VEL
LIN {X 0,Y 544.833,Z 538.128,A -85,B 0,C 180,E1 -3697.971,E2 -3697.971} C_VEL
LIN {X 0,Y 544.999,Z 530.174,A -85,B 0,C 180,E1 -3699.276,E2 -3699.276} C_VEL
LIN {X 0,Y 545.175,Z 521.853,A -85,B 0,C 180,E1 -3700.398,E2 -3700.398} C_VEL
LIN {X 0,Y 545.364,Z 512.028,A -85,B 0,C 180,E1 -3701.501,E2 -3701.501} C_VEL
LIN {X 0,Y 545.664,Z 500.646,A -85,B 0,C 180,E1 -3702.553,E2 -3702.553} C_VEL
LIN {X 0,Y 545.919,Z 488.103,A -85,B 0,C 180,E1 -3703.494,E2 -3703.494} C_VEL
LIN {X 0,Y 546.233,Z 475.641,A -85,B 0,C 180,E1 -3704.245,E2 -3704.245} C_VEL
LIN {X 0,Y 546.488,Z 461.697,A -85,B 0,C 180,E1 -3704.904,E2 -3704.904} C_VEL
LIN {X 0,Y 546.744,Z 448.343,A -85,B 0,C 180,E1 -3705.375,E2 -3705.375} C_VEL
LIN {X 0,Y 546.713,Z 437.3,A -85,B 0,C 180,E1 -3705.662,E2 -3705.662} C_VEL
LIN {X 0,Y 544.742,Z 427.806,A -85,B 0,C 180,E1 -3705.912,E2 -3705.912} C_VEL
LIN {X 0,Y 544.786,Z 420.842,A -85,B 0,C 180,E1 -3708.815,E2 -3708.815} C_VEL
LIN {X 0,Y 544.893,Z 413.772,A -85,B 0,C 180,E1 -3711.774,E2 -3711.774} C_VEL
LIN {X 0,Y 544.914,Z 407.718,A -85,B 0,C 180,E1 -3714.376,E2 -3714.376} C_VEL
LIN {X 0,Y 544.985,Z 401.411,A -85,B 0,C 180,E1 -3717.151,E2 -3717.151} C_VEL
LIN {X 0,Y 545.099,Z 394.515,A -85,B 0,C 180,E1 -3720.25,E2 -3720.25} C_VEL
LIN {X 0,Y 545.208,Z 388.424,A -85,B 0,C 180,E1 -3723.083,E2 -3723.083} C_VEL
LIN {X 0,Y 545.309,Z 381.62,A -85,B 0,C 180,E1 -3726.36,E2 -3726.36} C_VEL
LIN {X 0,Y 545.371,Z 377.914,A -85,B 0,C 180,E1 -3728.211,E2 -3728.211} C_VEL
LIN {X 0,Y 545.105,Z 375.215,A -85,B 0,C 180,E1 -3729.706,E2 -3729.706} C_VEL
LIN {X 0,Y 545.065,Z 375.218,A -85,B 0,C 180,E1 -3732.697,E2 -3732.697} C_VEL
LIN {X 0,Y 545.036,Z 375.218,A -85,B 0,C 180,E1 -3735.17,E2 -3735.17} C_VEL
LIN {X 0,Y 545.085,Z 375.216,A -85,B 0,C 180,E1 -3737.898,E2 -3737.898} C_VEL
LIN {X 0,Y 545.108,Z 375.209,A -85,B 0,C 180,E1 -3740.676,E2 -3740.676} C_VEL
LIN {X 0,Y 545.058,Z 375.214,A -85,B 0,C 180,E1 -3743.621,E2 -3743.621} C_VEL
LIN {X 0,Y 545.073,Z 375.214,A -85,B 0,C 180,E1 -3746.329,E2 -3746.329} C_VEL
LIN {X 0,Y 545.068,Z 375.216,A -85,B 0,C 180,E1 -3748.952,E2 -3748.952} C_VEL
LIN {X 0,Y 545.104,Z 375.208,A -85,B 0,C 180,E1 -3751.508,E2 -3751.508} C_VEL
LIN {X 0,Y 545.096,Z 375.21,A -85,B 0,C 180,E1 -3754.491,E2 -3754.491} C_VEL
LIN {X 0,Y 545.041,Z 375.221,A -85,B 0,C 180,E1 -3757.242,E2 -3757.242} C_VEL
LIN {X 0,Y 545.123,Z 375.21,A -85,B 0,C 180,E1 -3760.415,E2 -3760.415} C_VEL
LIN {X 0,Y 545.075,Z 375.214,A -85,B 0,C 180,E1 -3763.521,E2 -3763.521} C_VEL
LIN {X 0,Y 545.098,Z 375.209,A -85,B 0,C 180,E1 -3765.82,E2 -3765.82} C_VEL
LIN {X 0,Y 545.121,Z 375.209,A -85,B 0,C 180,E1 -3768.849,E2 -3768.849} C_VEL
LIN {X 0,Y 545.131,Z 375.21,A -85,B 0,C 180,E1 -3771.847,E2 -3771.847} C_VEL
LIN {X 0,Y 545.207,Z 375.197,A -85,B 0,C 180,E1 -3774.823,E2 -3774.823} C_VEL
LIN {X 0,Y 545.196,Z 375.196,A -85,B 0,C 180,E1 -3777.784,E2 -3777.784} C_VEL
LIN {X 0,Y 545.215,Z 375.194,A -85,B 0,C 180,E1 -3780.739,E2 -3780.739} C_VEL
LIN {X 0,Y 545.175,Z 375.201,A -85,B 0,C 180,E1 -3782.956,E2 -3782.956} C_VEL
LIN {X 0,Y 545.172,Z 375.199,A -85,B 0,C 180,E1 -3785.92,E2 -3785.92} C_VEL
LIN {X 0,Y 545.119,Z 375.205,A -85,B 0,C 180,E1 -3788.9,E2 -3788.9} C_VEL
LIN {X 0,Y 545.138,Z 375.204,A -85,B 0,C 180,E1 -3791.904,E2 -3791.904} C_VEL
LIN {X 0,Y 545.088,Z 375.212,A -85,B 0,C 180,E1 -3794.944,E2 -3794.944} C_VEL
LIN {X 0,Y 545.084,Z 375.214,A -85,B 0,C 180,E1 -3798.026,E2 -3798.026} C_VEL
LIN {X 0,Y 545.098,Z 375.208,A -85,B 0,C 180,E1 -3800.372,E2 -3800.372} C_VEL
LIN {X 0,Y 545.094,Z 375.209,A -85,B 0,C 180,E1 -3803.559,E2 -3803.559} C_VEL
LIN {X 0,Y 545.082,Z 375.216,A -85,B 0,C 180,E1 -3806.001,E2 -3806.001} C_VEL
LIN {X 0,Y 545.092,Z 375.21,A -85,B 0,C 180,E1 -3808.748,E2 -3808.748} C_VEL
LIN {X 0,Y 545.06,Z 375.213,A -85,B 0,C 180,E1 -3811.679,E2 -3811.679} C_VEL
LIN {X 0,Y 545.084,Z 375.211,A -85,B 0,C 180,E1 -3814.563,E2 -3814.563} C_VEL
LIN {X 0,Y 545.074,Z 375.214,A -85,B 0,C 180,E1 -3817.009,E2 -3817.009} C_VEL
LIN {X 0,Y 544.396,Z 375.302,A -85,B 0,C 180,E1 -3817.626,E2 -3817.626} C_VEL
LIN {X 0,Y 541.529,Z 375.657,A -85,B 0,C 180,E1 -3818.626,E2 -3818.626} C_VEL
LIN {X 0,Y 539.121,Z 375.954,A -85,B 0,C 180,E1 -3819.432,E2 -3819.432} C_VEL
LIN {X 0,Y 538.1,Z 376.081,A -85,B 0,C 180,E1 -3820.054,E2 -3820.054} C_VEL
LIN {X 0,Y 538.023,Z 376.089,A -85,B 0,C 180,E1 -3820.265,E2 -3820.265} C_VEL
LIN {X 0,Y 538.029,Z 376.089,A -85,B 0,C 180,E1 -3822.988,E2 -3822.988} C_VEL
LIN {X 0,Y 538.032,Z 376.09,A -85,B 0,C 180,E1 -3825.925,E2 -3825.925} C_VEL
LIN {X 0,Y 538.054,Z 376.088,A -85,B 0,C 180,E1 -3829.225,E2 -3829.225} C_VEL
LIN {X 0,Y 538.006,Z 376.098,A -85,B 0,C 180,E1 -3830.419,E2 -3830.419} C_VEL
LIN {X 0,Y 538.026,Z 376.511,A -85,B 0,C 180,E1 -3831.171,E2 -3831.171} C_VEL
LIN {X 0,Y 538.138,Z 379.661,A -85,B 0,C 180,E1 -3833.076,E2 -3833.076} C_VEL
LIN {X 0,Y 538.064,Z 384.379,A -85,B 0,C 180,E1 -3835.83,E2 -3835.83} C_VEL
LIN {X 0,Y 537.984,Z 389.09,A -85,B 0,C 180,E1 -3838.497,E2 -3838.497} C_VEL
LIN {X 0,Y 537.907,Z 393.797,A -85,B 0,C 180,E1 -3841.091,E2 -3841.091} C_VEL
LIN {X 0,Y 537.806,Z 398.501,A -85,B 0,C 180,E1 -3843.621,E2 -3843.621} C_VEL
LIN {X 0,Y 537.773,Z 403.308,A -85,B 0,C 180,E1 -3846.179,E2 -3846.179} C_VEL
LIN {X 0,Y 537.732,Z 407.828,A -85,B 0,C 180,E1 -3848.534,E2 -3848.534} C_VEL
LIN {X 0,Y 537.641,Z 414.086,A -85,B 0,C 180,E1 -3851.716,E2 -3851.716} C_VEL
LIN {X 0,Y 537.596,Z 418.529,A -85,B 0,C 180,E1 -3853.938,E2 -3853.938} C_VEL
LIN {X 0,Y 540.002,Z 429.933,A -85,B 0,C 180,E1 -3854.241,E2 -3854.241} C_VEL
LIN {X 0,Y 539.793,Z 443.173,A -85,B 0,C 180,E1 -3854.622,E2 -3854.622} C_VEL
LIN {X 0,Y 539.558,Z 457.218,A -85,B 0,C 180,E1 -3855.189,E2 -3855.189} C_VEL
LIN {X 0,Y 539.229,Z 469.9,A -85,B 0,C 180,E1 -3855.855,E2 -3855.855} C_VEL
LIN {X 0,Y 538.94,Z 481.533,A -85,B 0,C 180,E1 -3856.617,E2 -3856.617} C_VEL
LIN {X 0,Y 538.602,Z 493.381,A -85,B 0,C 180,E1 -3857.567,E2 -3857.567} C_VEL
LIN {X 0,Y 538.379,Z 503.597,A -85,B 0,C 180,E1 -3858.561,E2 -3858.561} C_VEL
LIN {X 0,Y 538.106,Z 512.986,A -85,B 0,C 180,E1 -3859.655,E2 -3859.655} C_VEL
LIN {X 0,Y 537.912,Z 521.114,A -85,B 0,C 180,E1 -3860.79,E2 -3860.79} C_VEL
LIN {X 0,Y 537.77,Z 528.895,A -85,B 0,C 180,E1 -3862.113,E2 -3862.113} C_VEL
LIN {X 0,Y 537.668,Z 535.101,A -85,B 0,C 180,E1 -3863.423,E2 -3863.423} C_VEL
LIN {X 0,Y 537.578,Z 540.053,A -85,B 0,C 180,E1 -3864.749,E2 -3864.749} C_VEL
LIN {X 0,Y 537.577,Z 544.214,A -85,B 0,C 180,E1 -3866.252,E2 -3866.252} C_VEL
LIN {X 0,Y 537.489,Z 546.938,A -85,B 0,C 180,E1 -3867.752,E2 -3867.752} C_VEL
LIN {X 0,Y 537.438,Z 548.307,A -85,B 0,C 180,E1 -3869.251,E2 -3869.251} C_VEL
LIN {X 0,Y 537.438,Z 548.353,A -85,B 0,C 180,E1 -3870.749,E2 -3870.749} C_VEL
LIN {X 0,Y 537.488,Z 547.068,A -85,B 0,C 180,E1 -3872.248,E2 -3872.248} C_VEL
LIN {X 0,Y 537.577,Z 544.422,A -85,B 0,C 180,E1 -3873.748,E2 -3873.748} C_VEL
LIN {X 0,Y 537.578,Z 540.349,A -85,B 0,C 180,E1 -3875.251,E2 -3875.251} C_VEL
LIN {X 0,Y 537.667,Z 534.72,A -85,B 0,C 180,E1 -3876.756,E2 -3876.756} C_VEL
LIN {X 0,Y 537.755,Z 528.366,A -85,B 0,C 180,E1 -3878.076,E2 -3878.076} C_VEL
LIN {X 0,Y 537.96,Z 520.466,A -85,B 0,C 180,E1 -3879.399,E2 -3879.399} C_VEL
LIN {X 0,Y 538.127,Z 512.203,A -85,B 0,C 180,E1 -3880.535,E2 -3880.535} C_VEL
LIN {X 0,Y 538.351,Z 503.095,A -85,B 0,C 180,E1 -3881.584,E2 -3881.584} C_VEL
LIN {X 0,Y 538.67,Z 492.248,A -85,B 0,C 180,E1 -3882.623,E2 -3882.623} C_VEL
LIN {X 0,Y 538.953,Z 480.155,A -85,B 0,C 180,E1 -3883.575,E2 -3883.575} C_VEL
LIN {X 0,Y 539.295,Z 468.201,A -85,B 0,C 180,E1 -3884.336,E2 -3884.336} C_VEL
LIN {X 0,Y 539.559,Z 455.012,A -85,B 0,C 180,E1 -3885.004,E2 -3885.004} C_VEL
LIN {X 0,Y 539.794,Z 440.793,A -85,B 0,C 180,E1 -3885.545,E2 -3885.545} C_VEL
LIN {X 0,Y 539.915,Z 429.413,A -85,B 0,C 180,E1 -3885.864,E2 -3885.864} C_VEL
LIN {X 0,Y 537.595,Z 418.526,A -85,B 0,C 180,E1 -3886.154,E2 -3886.154} C_VEL
LIN {X 0,Y 537.678,Z 412.738,A -85,B 0,C 180,E1 -3889.073,E2 -3889.073} C_VEL
LIN {X 0,Y 537.752,Z 406.518,A -85,B 0,C 180,E1 -3892.272,E2 -3892.272} C_VEL
LIN {X 0,Y 537.799,Z 401.802,A -85,B 0,C 180,E1 -3894.72,E2 -3894.72} C_VEL
LIN {X 0,Y 537.84,Z 396.923,A -85,B 0,C 180,E1 -3897.307,E2 -3897.307} C_VEL
LIN {X 0,Y 537.907,Z 392.388,A -85,B 0,C 180,E1 -3899.768,E2 -3899.768} C_VEL
LIN {X 0,Y 538.014,Z 387.681,A -85,B 0,C 180,E1 -3902.383,E2 -3902.383} C_VEL
LIN {X 0,Y 538.056,Z 382.971,A -85,B 0,C 180,E1 -3905.08,E2 -3905.08} C_VEL
LIN {X 0,Y 538.11,Z 378.235,A -85,B 0,C 180,E1 -3907.868,E2 -3907.868} C_VEL
LIN {X 0,Y 538.057,Z 376.663,A -85,B 0,C 180,E1 -3908.827,E2 -3908.827} C_VEL
LIN {X 0,Y 538.007,Z 376.1,A -85,B 0,C 180,E1 -3909.799,E2 -3909.799} C_VEL
LIN {X 0,Y 538.027,Z 376.094,A -85,B 0,C 180,E1 -3912.785,E2 -3912.785} C_VEL
LIN {X 0,Y 538.032,Z 376.091,A -85,B 0,C 180,E1 -3915.926,E2 -3915.926} C_VEL
LIN {X 0,Y 538.052,Z 376.09,A -85,B 0,C 180,E1 -3919.253,E2 -3919.253} C_VEL
LIN {X 0,Y 537.996,Z 376.093,A -85,B 0,C 180,E1 -3922.122,E2 -3922.122} C_VEL
LIN {X 0,Y 538.024,Z 376.09,A -85,B 0,C 180,E1 -3924.917,E2 -3924.917} C_VEL
LIN {X 0,Y 538.022,Z 376.095,A -85,B 0,C 180,E1 -3927.617,E2 -3927.617} C_VEL
LIN {X 0,Y 538.02,Z 376.09,A -85,B 0,C 180,E1 -3930.239,E2 -3930.239} C_VEL
LIN {X 0,Y 538.067,Z 376.087,A -85,B 0,C 180,E1 -3932.796,E2 -3932.796} C_VEL
LIN {X 0,Y 538.052,Z 376.087,A -85,B 0,C 180,E1 -3935.293,E2 -3935.293} C_VEL
LIN {X 0,Y 538.026,Z 376.091,A -85,B 0,C 180,E1 -3938.546,E2 -3938.546} C_VEL
LIN {X 0,Y 538.037,Z 376.09,A -85,B 0,C 180,E1 -3940.94,E2 -3940.94} C_VEL
LIN {X 0,Y 538.028,Z 376.09,A -85,B 0,C 180,E1 -3943.299,E2 -3943.299} C_VEL
LIN {X 0,Y 538.068,Z 376.088,A -85,B 0,C 180,E1 -3945.631,E2 -3945.631} C_VEL
LIN {X 0,Y 538.081,Z 376.088,A -85,B 0,C 180,E1 -3948.702,E2 -3948.702} C_VEL
LIN {X 0,Y 538.089,Z 376.085,A -85,B 0,C 180,E1 -3951.74,E2 -3951.74} C_VEL
LIN {X 0,Y 538.165,Z 376.073,A -85,B 0,C 180,E1 -3954.755,E2 -3954.755} C_VEL
LIN {X 0,Y 538.168,Z 376.072,A -85,B 0,C 180,E1 -3957.755,E2 -3957.755} C_VEL
LIN {X 0,Y 538.186,Z 376.069,A -85,B 0,C 180,E1 -3960.748,E2 -3960.748} C_VEL
LIN {X 0,Y 538.143,Z 376.077,A -85,B 0,C 180,E1 -3962.994,E2 -3962.994} C_VEL
LIN {X 0,Y 538.126,Z 376.077,A -85,B 0,C 180,E1 -3965.997,E2 -3965.997} C_VEL
LIN {X 0,Y 538.066,Z 376.084,A -85,B 0,C 180,E1 -3969.018,E2 -3969.018} C_VEL
LIN {X 0,Y 538.087,Z 376.082,A -85,B 0,C 180,E1 -3972.062,E2 -3972.062} C_VEL
LIN {X 0,Y 538.049,Z 376.087,A -85,B 0,C 180,E1 -3975.144,E2 -3975.144} C_VEL
LIN {X 0,Y 538.037,Z 376.089,A -85,B 0,C 180,E1 -3978.27,E2 -3978.27} C_VEL
LIN {X 0,Y 538.043,Z 376.088,A -85,B 0,C 180,E1 -3980.651,E2 -3980.651} C_VEL
LIN {X 0,Y 538.028,Z 376.089,A -85,B 0,C 180,E1 -3983.887,E2 -3983.887} C_VEL
LIN {X 0,Y 538.044,Z 376.088,A -85,B 0,C 180,E1 -3986.367,E2 -3986.367} C_VEL
LIN {X 0,Y 538.034,Z 376.091,A -85,B 0,C 180,E1 -3988.933,E2 -3988.933} C_VEL
LIN {X 0,Y 538.013,Z 376.091,A -85,B 0,C 180,E1 -3991.887,E2 -3991.887} C_VEL
LIN {X 0,Y 538.034,Z 376.089,A -85,B 0,C 180,E1 -3994.621,E2 -3994.621} C_VEL
LIN {X 0,Y 538.011,Z 376.097,A -85,B 0,C 180,E1 -3997.17,E2 -3997.17} C_VEL
LIN {X 0,Y 538.057,Z 376.087,A -85,B 0,C 180,E1 -3999.794,E2 -3999.794} C_VEL
LIN {X 0,Y 538.021,Z 376.091,A -85,B 0,C 180,E1 -4002.786,E2 -4002.786} C_VEL
LIN {X 0,Y 538.031,Z 376.091,A -85,B 0,C 180,E1 -4005.925,E2 -4005.925} C_VEL
LIN {X 0,Y 538.054,Z 376.089,A -85,B 0,C 180,E1 -4009.252,E2 -4009.252} C_VEL
LIN {X 0,Y 538.092,Z 376.293,A -85,B 0,C 180,E1 -4010.34,E2 -4010.34} C_VEL
LIN {X 0,Y 538.325,Z 379.746,A -85,B 0,C 180,E1 -4012.15,E2 -4012.15} C_VEL
LIN {X 0,Y 538.219,Z 385.315,A -85,B 0,C 180,E1 -4014.932,E2 -4014.932} C_VEL
LIN {X 0,Y 538.134,Z 390.896,A -85,B 0,C 180,E1 -4017.625,E2 -4017.625} C_VEL
LIN {X 0,Y 538.031,Z 396.487,A -85,B 0,C 180,E1 -4020.24,E2 -4020.24} C_VEL
LIN {X 0,Y 537.941,Z 402.108,A -85,B 0,C 180,E1 -4022.789,E2 -4022.789} C_VEL
LIN {X 0,Y 537.865,Z 407.725,A -85,B 0,C 180,E1 -4025.283,E2 -4025.283} C_VEL
LIN {X 0,Y 537.815,Z 415.206,A -85,B 0,C 180,E1 -4028.537,E2 -4028.537} C_VEL
LIN {X 0,Y 537.744,Z 420.812,A -85,B 0,C 180,E1 -4030.929,E2 -4030.929} C_VEL
LIN {X 0,Y 537.663,Z 427.849,A -85,B 0,C 180,E1 -4033.891,E2 -4033.891} C_VEL
LIN {X 0,Y 540.028,Z 439.801,A -85,B 0,C 180,E1 -4034.193,E2 -4034.193} C_VEL
LIN {X 0,Y 539.77,Z 453.545,A -85,B 0,C 180,E1 -4034.59,E2 -4034.59} C_VEL
LIN {X 0,Y 539.531,Z 466.161,A -85,B 0,C 180,E1 -4035.092,E2 -4035.092} C_VEL
LIN {X 0,Y 539.259,Z 479.052,A -85,B 0,C 180,E1 -4035.759,E2 -4035.759} C_VEL
LIN {X 0,Y 538.956,Z 490.843,A -85,B 0,C 180,E1 -4036.521,E2 -4036.521} C_VEL
LIN {X 0,Y 538.618,Z 502.814,A -85,B 0,C 180,E1 -4037.471,E2 -4037.471} C_VEL
LIN {X 0,Y 538.388,Z 513.966,A -85,B 0,C 180,E1 -4038.555,E2 -4038.555} C_VEL
LIN {X 0,Y 538.096,Z 523.337,A -85,B 0,C 180,E1 -4039.654,E2 -4039.654} C_VEL
LIN {X 0,Y 537.919,Z 531.405,A -85,B 0,C 180,E1 -4040.79,E2 -4040.79} C_VEL
LIN {X 0,Y 537.763,Z 539.134,A -85,B 0,C 180,E1 -4042.113,E2 -4042.113} C_VEL
LIN {X 0,Y 537.686,Z 545.218,A -85,B 0,C 180,E1 -4043.406,E2 -4043.406} C_VEL
LIN {X 0,Y 537.579,Z 550.2,A -85,B 0,C 180,E1 -4044.749,E2 -4044.749} C_VEL
LIN {X 0,Y 537.576,Z 554.316,A -85,B 0,C 180,E1 -4046.252,E2 -4046.252} C_VEL
LIN {X 0,Y 537.489,Z 557.002,A -85,B 0,C 180,E1 -4047.752,E2 -4047.752} C_VEL
LIN {X 0,Y 537.439,Z 558.333,A -85,B 0,C 180,E1 -4049.251,E2 -4049.251} C_VEL
LIN {X 0,Y 537.439,Z 558.334,A -85,B 0,C 180,E1 -4050.749,E2 -4050.749} C_VEL
LIN {X 0,Y 537.489,Z 557.004,A -85,B 0,C 180,E1 -4052.248,E2 -4052.248} C_VEL
LIN {X 0,Y 537.576,Z 554.32,A -85,B 0,C 180,E1 -4053.748,E2 -4053.748} C_VEL
LIN {X 0,Y 537.579,Z 550.202,A -85,B 0,C 180,E1 -4055.251,E2 -4055.251} C_VEL
LIN {X 0,Y 537.672,Z 545.273,A -85,B 0,C 180,E1 -4056.581,E2 -4056.581} C_VEL
LIN {X 0,Y 537.763,Z 539.135,A -85,B 0,C 180,E1 -4057.887,E2 -4057.887} C_VEL
LIN {X 0,Y 537.918,Z 531.406,A -85,B 0,C 180,E1 -4059.21,E2 -4059.21} C_VEL
LIN {X 0,Y 538.096,Z 523.338,A -85,B 0,C 180,E1 -4060.346,E2 -4060.346} C_VEL
LIN {X 0,Y 538.363,Z 514.035,A -85,B 0,C 180,E1 -4061.438,E2 -4061.438} C_VEL
LIN {X 0,Y 538.618,Z 502.815,A -85,B 0,C 180,E1 -4062.529,E2 -4062.529} C_VEL
LIN {X 0,Y 538.956,Z 490.847,A -85,B 0,C 180,E1 -4063.479,E2 -4063.479} C_VEL
LIN {X 0,Y 539.259,Z 479.057,A -85,B 0,C 180,E1 -4064.24,E2 -4064.24} C_VEL
LIN {X 0,Y 539.522,Z 466.156,A -85,B 0,C 180,E1 -4064.908,E2 -4064.908} C_VEL
LIN {X 0,Y 539.763,Z 453.035,A -85,B 0,C 180,E1 -4065.429,E2 -4065.429} C_VEL
LIN {X 0,Y 539.9,Z 438.475,A -85,B 0,C 180,E1 -4065.839,E2 -4065.839} C_VEL
LIN {X 0,Y 537.668,Z 427.806,A -85,B 0,C 180,E1 -4066.127,E2 -4066.127} C_VEL
LIN {X 0,Y 537.744,Z 420.777,A -85,B 0,C 180,E1 -4069.071,E2 -4069.071} C_VEL
LIN {X 0,Y 537.831,Z 414.086,A -85,B 0,C 180,E1 -4071.909,E2 -4071.909} C_VEL
LIN {X 0,Y 537.859,Z 407.674,A -85,B 0,C 180,E1 -4074.717,E2 -4074.717} C_VEL
LIN {X 0,Y 537.939,Z 401.827,A -85,B 0,C 180,E1 -4077.327,E2 -4077.327} C_VEL
LIN {X 0,Y 538.045,Z 395.005,A -85,B 0,C 180,E1 -4080.447,E2 -4080.447} C_VEL
LIN {X 0,Y 538.188,Z 388.943,A -85,B 0,C 180,E1 -4083.306,E2 -4083.306} C_VEL
LIN {X 0,Y 538.301,Z 383.454,A -85,B 0,C 180,E1 -4085.981,E2 -4085.981} C_VEL
LIN {X 0,Y 538.286,Z 377.891,A -85,B 0,C 180,E1 -4088.807,E2 -4088.807} C_VEL
LIN {X 0,Y 538.078,Z 376.091,A -85,B 0,C 180,E1 -4089.792,E2 -4089.792} C_VEL
LIN {X 0,Y 538.028,Z 376.095,A -85,B 0,C 180,E1 -4092.988,E2 -4092.988} C_VEL
LIN {X 0,Y 538.004,Z 376.099,A -85,B 0,C 180,E1 -4096.184,E2 -4096.184} C_VEL
LIN {X 0,Y 538.08,Z 376.087,A -85,B 0,C 180,E1 -4099.249,E2 -4099.249} C_VEL
LIN {X 0,Y 538.003,Z 376.093,A -85,B 0,C 180,E1 -4102.123,E2 -4102.123} C_VEL
LIN {X 0,Y 538.022,Z 376.091,A -85,B 0,C 180,E1 -4104.917,E2 -4104.917} C_VEL
LIN {X 0,Y 538.028,Z 376.095,A -85,B 0,C 180,E1 -4107.618,E2 -4107.618} C_VEL
LIN {X 0,Y 538.019,Z 376.091,A -85,B 0,C 180,E1 -4110.239,E2 -4110.239} C_VEL
LIN {X 0,Y 538.065,Z 376.086,A -85,B 0,C 180,E1 -4112.796,E2 -4112.796} C_VEL
LIN {X 0,Y 538.03,Z 376.091,A -85,B 0,C 180,E1 -4115.292,E2 -4115.292} C_VEL
LIN {X 0,Y 538.017,Z 376.09,A -85,B 0,C 180,E1 -4118.042,E2 -4118.042} C_VEL
LIN {X 0,Y 538.041,Z 376.089,A -85,B 0,C 180,E1 -4120.94,E2 -4120.94} C_VEL
LIN {X 0,Y 538.027,Z 376.09,A -85,B 0,C 180,E1 -4123.299,E2 -4123.299} C_VEL
LIN {X 0,Y 538.067,Z 376.087,A -85,B 0,C 180,E1 -4125.631,E2 -4125.631} C_VEL
LIN {X 0,Y 538.08,Z 376.087,A -85,B 0,C 180,E1 -4128.702,E2 -4128.702} C_VEL
LIN {X 0,Y 538.088,Z 376.086,A -85,B 0,C 180,E1 -4131.74,E2 -4131.74} C_VEL
LIN {X 0,Y 538.164,Z 376.074,A -85,B 0,C 180,E1 -4134.755,E2 -4134.755} C_VEL
LIN {X 0,Y 538.169,Z 376.071,A -85,B 0,C 180,E1 -4137.755,E2 -4137.755} C_VEL
LIN {X 0,Y 538.185,Z 376.069,A -85,B 0,C 180,E1 -4140.748,E2 -4140.748} C_VEL
LIN {X 0,Y 538.141,Z 376.078,A -85,B 0,C 180,E1 -4142.995,E2 -4142.995} C_VEL
LIN {X 0,Y 538.126,Z 376.078,A -85,B 0,C 180,E1 -4145.997,E2 -4145.997} C_VEL
LIN {X 0,Y 538.07,Z 376.083,A -85,B 0,C 180,E1 -4149.018,E2 -4149.018} C_VEL
LIN {X 0,Y 538.086,Z 376.082,A -85,B 0,C 180,E1 -4152.063,E2 -4152.063} C_VEL
LIN {X 0,Y 538.048,Z 376.087,A -85,B 0,C 180,E1 -4155.144,E2 -4155.144} C_VEL
LIN {X 0,Y 538.036,Z 376.09,A -85,B 0,C 180,E1 -4158.27,E2 -4158.27} C_VEL
LIN {X 0,Y 538.042,Z 376.088,A -85,B 0,C 180,E1 -4160.651,E2 -4160.651} C_VEL
LIN {X 0,Y 538.027,Z 376.09,A -85,B 0,C 180,E1 -4163.887,E2 -4163.887} C_VEL
LIN {X 0,Y 538.044,Z 376.089,A -85,B 0,C 180,E1 -4166.367,E2 -4166.367} C_VEL
LIN {X 0,Y 538.033,Z 376.091,A -85,B 0,C 180,E1 -4168.934,E2 -4168.934} C_VEL
LIN {X 0,Y 538.012,Z 376.091,A -85,B 0,C 180,E1 -4171.887,E2 -4171.887} C_VEL
LIN {X 0,Y 538.034,Z 376.089,A -85,B 0,C 180,E1 -4174.621,E2 -4174.621} C_VEL
LIN {X 0,Y 538.026,Z 376.094,A -85,B 0,C 180,E1 -4177.173,E2 -4177.173} C_VEL
LIN {X 0,Y 538.023,Z 376.089,A -85,B 0,C 180,E1 -4180.265,E2 -4180.265} C_VEL
LIN {X 0,Y 537.373,Z 376.175,A -85,B 0,C 180,E1 -4180.89,E2 -4180.89} C_VEL
LIN {X 0,Y 534.519,Z 376.533,A -85,B 0,C 180,E1 -4181.905,E2 -4181.905} C_VEL
LIN {X 0,Y 532.094,Z 376.835,A -85,B 0,C 180,E1 -4182.722,E2 -4182.722} C_VEL
LIN {X 0,Y 531.046,Z 376.963,A -85,B 0,C 180,E1 -4183.353,E2 -4183.353} C_VEL
LIN {X 0,Y 530.959,Z 376.972,A -85,B 0,C 180,E1 -4183.567,E2 -4183.567} C_VEL
LIN {X 0,Y 530.969,Z 376.97,A -85,B 0,C 180,E1 -4186.506,E2 -4186.506} C_VEL
LIN {X 0,Y 530.992,Z 376.97,A -85,B 0,C 180,E1 -4188.976,E2 -4188.976} C_VEL
LIN {X 0,Y 530.967,Z 376.974,A -85,B 0,C 180,E1 -4190.555,E2 -4190.555} C_VEL
LIN {X 0,Y 531.034,Z 378.116,A -85,B 0,C 180,E1 -4191.536,E2 -4191.536} C_VEL
LIN {X 0,Y 531.074,Z 381.894,A -85,B 0,C 180,E1 -4193.828,E2 -4193.828} C_VEL
LIN {X 0,Y 531.008,Z 386.441,A -85,B 0,C 180,E1 -4196.493,E2 -4196.493} C_VEL
LIN {X 0,Y 530.891,Z 391.501,A -85,B 0,C 180,E1 -4199.371,E2 -4199.371} C_VEL
LIN {X 0,Y 530.824,Z 395.406,A -85,B 0,C 180,E1 -4201.534,E2 -4201.534} C_VEL
LIN {X 0,Y 530.757,Z 400.356,A -85,B 0,C 180,E1 -4204.214,E2 -4204.214} C_VEL
LIN {X 0,Y 530.685,Z 404.79,A -85,B 0,C 180,E1 -4206.591,E2 -4206.591} C_VEL
LIN {X 0,Y 530.624,Z 409.46,A -85,B 0,C 180,E1 -4209.047,E2 -4209.047} C_VEL
LIN {X 0,Y 530.561,Z 414.141,A -85,B 0,C 180,E1 -4211.463,E2 -4211.463} C_VEL
LIN {X 0,Y 530.542,Z 418.587,A -85,B 0,C 180,E1 -4213.725,E2 -4213.725} C_VEL
LIN {X 0,Y 533.13,Z 431.019,A -85,B 0,C 180,E1 -4214.06,E2 -4214.06} C_VEL
LIN {X 0,Y 532.947,Z 445.311,A -85,B 0,C 180,E1 -4214.498,E2 -4214.498} C_VEL
LIN {X 0,Y 532.619,Z 459.229,A -85,B 0,C 180,E1 -4215.09,E2 -4215.09} C_VEL
LIN {X 0,Y 532.276,Z 471.49,A -85,B 0,C 180,E1 -4215.764,E2 -4215.764} C_VEL
LIN {X 0,Y 531.911,Z 484.12,A -85,B 0,C 180,E1 -4216.631,E2 -4216.631} C_VEL
LIN {X 0,Y 531.568,Z 495.524,A -85,B 0,C 180,E1 -4217.594,E2 -4217.594} C_VEL
LIN {X 0,Y 531.325,Z 504.978,A -85,B 0,C 180,E1 -4218.556,E2 -4218.556} C_VEL
LIN {X 0,Y 531.028,Z 514.475,A -85,B 0,C 180,E1 -4219.708,E2 -4219.708} C_VEL
LIN {X 0,Y 530.811,Z 523.541,A -85,B 0,C 180,E1 -4221.05,E2 -4221.05} C_VEL
LIN {X 0,Y 530.643,Z 530.841,A -85,B 0,C 180,E1 -4222.389,E2 -4222.389} C_VEL
LIN {X 0,Y 530.559,Z 537.4,A -85,B 0,C 180,E1 -4223.917,E2 -4223.917} C_VEL
LIN {X 0,Y 530.449,Z 542.321,A -85,B 0,C 180,E1 -4225.441,E2 -4225.441} C_VEL
LIN {X 0,Y 530.453,Z 545.751,A -85,B 0,C 180,E1 -4226.962,E2 -4226.962} C_VEL
LIN {X 0,Y 530.36,Z 547.79,A -85,B 0,C 180,E1 -4228.481,E2 -4228.481} C_VEL
LIN {X 0,Y 530.342,Z 548.497,A -85,B 0,C 180,E1 -4230,E2 -4230} C_VEL
LIN {X 0,Y 530.358,Z 547.877,A -85,B 0,C 180,E1 -4231.519,E2 -4231.519} C_VEL
LIN {X 0,Y 530.452,Z 545.917,A -85,B 0,C 180,E1 -4233.038,E2 -4233.038} C_VEL
LIN {X 0,Y 530.449,Z 542.569,A -85,B 0,C 180,E1 -4234.56,E2 -4234.56} C_VEL
LIN {X 0,Y 530.537,Z 537.736,A -85,B 0,C 180,E1 -4236.083,E2 -4236.083} C_VEL
LIN {X 0,Y 530.587,Z 533.076,A -85,B 0,C 180,E1 -4237.229,E2 -4237.229} C_VEL
LIN {X 0,Y 530.774,Z 526.295,A -85,B 0,C 180,E1 -4238.567,E2 -4238.567} C_VEL
LIN {X 0,Y 530.915,Z 517.872,A -85,B 0,C 180,E1 -4239.909,E2 -4239.909} C_VEL
LIN {X 0,Y 531.221,Z 509.084,A -85,B 0,C 180,E1 -4241.06,E2 -4241.06} C_VEL
LIN {X 0,Y 531.472,Z 498.437,A -85,B 0,C 180,E1 -4242.215,E2 -4242.215} C_VEL
LIN {X 0,Y 531.818,Z 487.674,A -85,B 0,C 180,E1 -4243.177,E2 -4243.177} C_VEL
LIN {X 0,Y 532.161,Z 475.901,A -85,B 0,C 180,E1 -4244.044,E2 -4244.044} C_VEL
LIN {X 0,Y 532.529,Z 462.925,A -85,B 0,C 180,E1 -4244.815,E2 -4244.815} C_VEL
LIN {X 0,Y 532.856,Z 449.93,A -85,B 0,C 180,E1 -4245.418,E2 -4245.418} C_VEL
LIN {X 0,Y 533.089,Z 435.517,A -85,B 0,C 180,E1 -4245.911,E2 -4245.911} C_VEL
LIN {X 0,Y 533.042,Z 430.25,A -85,B 0,C 180,E1 -4246.054,E2 -4246.054} C_VEL
LIN {X 0,Y 530.556,Z 418.591,A -85,B 0,C 180,E1 -4246.374,E2 -4246.374} C_VEL
LIN {X 0,Y 530.605,Z 412.809,A -85,B 0,C 180,E1 -4249.338,E2 -4249.338} C_VEL
LIN {X 0,Y 530.667,Z 407.651,A -85,B 0,C 180,E1 -4252.018,E2 -4252.018} C_VEL
LIN {X 0,Y 530.724,Z 401.846,A -85,B 0,C 180,E1 -4255.072,E2 -4255.072} C_VEL
LIN {X 0,Y 530.789,Z 397.137,A -85,B 0,C 180,E1 -4257.608,E2 -4257.608} C_VEL
LIN {X 0,Y 530.864,Z 392.425,A -85,B 0,C 180,E1 -4260.204,E2 -4260.204} C_VEL
LIN {X 0,Y 530.967,Z 387.714,A -85,B 0,C 180,E1 -4262.867,E2 -4262.867} C_VEL
LIN {X 0,Y 531.042,Z 382.991,A -85,B 0,C 180,E1 -4265.613,E2 -4265.613} C_VEL
LIN {X 0,Y 531.101,Z 379.843,A -85,B 0,C 180,E1 -4267.497,E2 -4267.497} C_VEL
LIN {X 0,Y 531.045,Z 377.94,A -85,B 0,C 180,E1 -4268.664,E2 -4268.664} C_VEL
LIN {X 0,Y 530.971,Z 376.975,A -85,B 0,C 180,E1 -4269.445,E2 -4269.445} C_VEL
LIN {X 0,Y 530.984,Z 376.968,A -85,B 0,C 180,E1 -4272.456,E2 -4272.456} C_VEL
LIN {X 0,Y 530.991,Z 376.967,A -85,B 0,C 180,E1 -4275.621,E2 -4275.621} C_VEL
LIN {X 0,Y 531,Z 376.966,A -85,B 0,C 180,E1 -4278.565,E2 -4278.565} C_VEL
LIN {X 0,Y 530.96,Z 376.971,A -85,B 0,C 180,E1 -4281.529,E2 -4281.529} C_VEL
LIN {X 0,Y 530.986,Z 376.972,A -85,B 0,C 180,E1 -4284.382,E2 -4284.382} C_VEL
LIN {X 0,Y 530.97,Z 376.969,A -85,B 0,C 180,E1 -4287.133,E2 -4287.133} C_VEL
LIN {X 0,Y 530.973,Z 376.968,A -85,B 0,C 180,E1 -4289.803,E2 -4289.803} C_VEL
LIN {X 0,Y 531.018,Z 376.968,A -85,B 0,C 180,E1 -4292.467,E2 -4292.467} C_VEL
LIN {X 0,Y 531.009,Z 376.963,A -85,B 0,C 180,E1 -4294.943,E2 -4294.943} C_VEL
LIN {X 0,Y 530.975,Z 376.968,A -85,B 0,C 180,E1 -4298.247,E2 -4298.247} C_VEL
LIN {X 0,Y 530.997,Z 376.97,A -85,B 0,C 180,E1 -4300.677,E2 -4300.677} C_VEL
LIN {X 0,Y 530.989,Z 376.966,A -85,B 0,C 180,E1 -4303.071,E2 -4303.071} C_VEL
LIN {X 0,Y 531.045,Z 376.965,A -85,B 0,C 180,E1 -4305.436,E2 -4305.436} C_VEL
LIN {X 0,Y 531.041,Z 376.964,A -85,B 0,C 180,E1 -4308.55,E2 -4308.55} C_VEL
LIN {X 0,Y 531.059,Z 376.959,A -85,B 0,C 180,E1 -4311.629,E2 -4311.629} C_VEL
LIN {X 0,Y 531.124,Z 376.95,A -85,B 0,C 180,E1 -4314.685,E2 -4314.685} C_VEL
LIN {X 0,Y 531.14,Z 376.947,A -85,B 0,C 180,E1 -4317.725,E2 -4317.725} C_VEL
LIN {X 0,Y 531.156,Z 376.944,A -85,B 0,C 180,E1 -4320.758,E2 -4320.758} C_VEL
LIN {X 0,Y 531.11,Z 376.954,A -85,B 0,C 180,E1 -4323.034,E2 -4323.034} C_VEL
LIN {X 0,Y 531.086,Z 376.954,A -85,B 0,C 180,E1 -4326.077,E2 -4326.077} C_VEL
LIN {X 0,Y 531.028,Z 376.961,A -85,B 0,C 180,E1 -4329.138,E2 -4329.138} C_VEL
LIN {X 0,Y 531.044,Z 376.959,A -85,B 0,C 180,E1 -4332.225,E2 -4332.225} C_VEL
LIN {X 0,Y 530.999,Z 376.965,A -85,B 0,C 180,E1 -4335.35,E2 -4335.35} C_VEL
LIN {X 0,Y 530.996,Z 376.965,A -85,B 0,C 180,E1 -4338.521,E2 -4338.521} C_VEL
LIN {X 0,Y 531.004,Z 376.968,A -85,B 0,C 180,E1 -4340.938,E2 -4340.938} C_VEL
LIN {X 0,Y 530.984,Z 376.97,A -85,B 0,C 180,E1 -4344.224,E2 -4344.224} C_VEL
LIN {X 0,Y 531.007,Z 376.963,A -85,B 0,C 180,E1 -4346.744,E2 -4346.744} C_VEL
LIN {X 0,Y 530.985,Z 376.97,A -85,B 0,C 180,E1 -4349.322,E2 -4349.322} C_VEL
LIN {X 0,Y 530.968,Z 376.971,A -85,B 0,C 180,E1 -4352.1,E2 -4352.1} C_VEL
LIN {X 0,Y 530.992,Z 376.966,A -85,B 0,C 180,E1 -4354.854,E2 -4354.854} C_VEL
LIN {X 0,Y 530.97,Z 376.973,A -85,B 0,C 180,E1 -4357.507,E2 -4357.507} C_VEL
LIN {X 0,Y 531.029,Z 376.967,A -85,B 0,C 180,E1 -4360.429,E2 -4360.429} C_VEL
LIN {X 0,Y 530.956,Z 376.974,A -85,B 0,C 180,E1 -4363.496,E2 -4363.496} C_VEL
LIN {X 0,Y 530.967,Z 376.971,A -85,B 0,C 180,E1 -4366.505,E2 -4366.505} C_VEL
LIN {X 0,Y 531,Z 376.968,A -85,B 0,C 180,E1 -4369.569,E2 -4369.569} C_VEL
LIN {X 0,Y 531.061,Z 377.069,A -85,B 0,C 180,E1 -4370.136,E2 -4370.136} C_VEL
LIN {X 0,Y 531.322,Z 379.725,A -85,B 0,C 180,E1 -4371.56,E2 -4371.56} C_VEL
LIN {X 0,Y 531.235,Z 385.286,A -85,B 0,C 180,E1 -4374.401,E2 -4374.401} C_VEL
LIN {X 0,Y 531.117,Z 390.863,A -85,B 0,C 180,E1 -4377.144,E2 -4377.144} C_VEL
LIN {X 0,Y 530.986,Z 396.451,A -85,B 0,C 180,E1 -4379.804,E2 -4379.804} C_VEL
LIN {X 0,Y 530.894,Z 402.269,A -85,B 0,C 180,E1 -4382.492,E2 -4382.492} C_VEL
LIN {X 0,Y 530.801,Z 407.69,A -85,B 0,C 180,E1 -4384.932,E2 -4384.932} C_VEL
LIN {X 0,Y 530.752,Z 415.172,A -85,B 0,C 180,E1 -4388.237,E2 -4388.237} C_VEL
LIN {X 0,Y 530.684,Z 420.779,A -85,B 0,C 180,E1 -4390.665,E2 -4390.665} C_VEL
LIN {X 0,Y 530.607,Z 427.824,A -85,B 0,C 180,E1 -4393.671,E2 -4393.671} C_VEL
LIN {X 0,Y 533.193,Z 441.065,A -85,B 0,C 180,E1 -4394.019,E2 -4394.019} C_VEL
LIN {X 0,Y 532.904,Z 453.868,A -85,B 0,C 180,E1 -4394.399,E2 -4394.399} C_VEL
LIN {X 0,Y 532.638,Z 466.153,A -85,B 0,C 180,E1 -4394.894,E2 -4394.894} C_VEL
LIN {X 0,Y 532.362,Z 479.051,A -85,B 0,C 180,E1 -4395.571,E2 -4395.571} C_VEL
LIN {X 0,Y 531.989,Z 492.133,A -85,B 0,C 180,E1 -4396.438,E2 -4396.438} C_VEL
LIN {X 0,Y 531.628,Z 503.882,A -85,B 0,C 180,E1 -4397.401,E2 -4397.401} C_VEL
LIN {X 0,Y 531.372,Z 514.245,A -85,B 0,C 180,E1 -4398.433,E2 -4398.433} C_VEL
LIN {X 0,Y 531.087,Z 523.336,A -85,B 0,C 180,E1 -4399.516,E2 -4399.516} C_VEL
LIN {X 0,Y 530.889,Z 531.404,A -85,B 0,C 180,E1 -4400.667,E2 -4400.667} C_VEL
LIN {X 0,Y 530.684,Z 539.133,A -85,B 0,C 180,E1 -4402.007,E2 -4402.007} C_VEL
LIN {X 0,Y 530.611,Z 545.592,A -85,B 0,C 180,E1 -4403.406,E2 -4403.406} C_VEL
LIN {X 0,Y 530.514,Z 550.2,A -85,B 0,C 180,E1 -4404.679,E2 -4404.679} C_VEL
LIN {X 0,Y 530.497,Z 554.316,A -85,B 0,C 180,E1 -4406.202,E2 -4406.202} C_VEL
LIN {X 0,Y 530.41,Z 557.002,A -85,B 0,C 180,E1 -4407.722,E2 -4407.722} C_VEL
LIN {X 0,Y 530.341,Z 558.334,A -85,B 0,C 180,E1 -4409.241,E2 -4409.241} C_VEL
LIN {X 0,Y 530.341,Z 558.334,A -85,B 0,C 180,E1 -4410.759,E2 -4410.759} C_VEL
LIN {X 0,Y 530.41,Z 557.005,A -85,B 0,C 180,E1 -4412.278,E2 -4412.278} C_VEL
LIN {X 0,Y 530.497,Z 554.32,A -85,B 0,C 180,E1 -4413.798,E2 -4413.798} C_VEL
LIN {X 0,Y 530.514,Z 550.202,A -85,B 0,C 180,E1 -4415.321,E2 -4415.321} C_VEL
LIN {X 0,Y 530.573,Z 544.526,A -85,B 0,C 180,E1 -4416.847,E2 -4416.847} C_VEL
LIN {X 0,Y 530.709,Z 538.127,A -85,B 0,C 180,E1 -4418.184,E2 -4418.184} C_VEL
LIN {X 0,Y 530.928,Z 530.174,A -85,B 0,C 180,E1 -4419.524,E2 -4419.524} C_VEL
LIN {X 0,Y 531.13,Z 521.852,A -85,B 0,C 180,E1 -4420.676,E2 -4420.676} C_VEL
LIN {X 0,Y 531.454,Z 511.354,A -85,B 0,C 180,E1 -4421.879,E2 -4421.879} C_VEL
LIN {X 0,Y 531.711,Z 500.649,A -85,B 0,C 180,E1 -4422.888,E2 -4422.888} C_VEL
LIN {X 0,Y 532.089,Z 488.1,A -85,B 0,C 180,E1 -4423.851,E2 -4423.851} C_VEL
LIN {X 0,Y 532.465,Z 475.637,A -85,B 0,C 180,E1 -4424.621,E2 -4424.621} C_VEL
LIN {X 0,Y 532.764,Z 461.682,A -85,B 0,C 180,E1 -4425.297,E2 -4425.297} C_VEL
LIN {X 0,Y 533.047,Z 447.661,A -85,B 0,C 180,E1 -4425.801,E2 -4425.801} C_VEL
LIN {X 0,Y 532.994,Z 439.285,A -85,B 0,C 180,E1 -4426.032,E2 -4426.032} C_VEL
LIN {X 0,Y 530.601,Z 427.75,A -85,B 0,C 180,E1 -4426.348,E2 -4426.348} C_VEL
LIN {X 0,Y 530.683,Z 420.704,A -85,B 0,C 180,E1 -4429.334,E2 -4429.334} C_VEL
LIN {X 0,Y 530.752,Z 414.438,A -85,B 0,C 180,E1 -4432.042,E2 -4432.042} C_VEL
LIN {X 0,Y 530.791,Z 407.629,A -85,B 0,C 180,E1 -4435.068,E2 -4435.068} C_VEL
LIN {X 0,Y 530.897,Z 402.039,A -85,B 0,C 180,E1 -4437.602,E2 -4437.602} C_VEL
LIN {X 0,Y 530.986,Z 396.45,A -85,B 0,C 180,E1 -4440.196,E2 -4440.196} C_VEL
LIN {X 0,Y 531.117,Z 390.862,A -85,B 0,C 180,E1 -4442.856,E2 -4442.856} C_VEL
LIN {X 0,Y 531.234,Z 385.288,A -85,B 0,C 180,E1 -4445.598,E2 -4445.598} C_VEL
LIN {X 0,Y 531.32,Z 379.723,A -85,B 0,C 180,E1 -4448.44,E2 -4448.44} C_VEL
LIN {X 0,Y 531.029,Z 376.969,A -85,B 0,C 180,E1 -4449.955,E2 -4449.955} C_VEL
LIN {X 0,Y 530.982,Z 376.97,A -85,B 0,C 180,E1 -4452.456,E2 -4452.456} C_VEL
LIN {X 0,Y 530.978,Z 376.969,A -85,B 0,C 180,E1 -4455.622,E2 -4455.622} C_VEL
LIN {X 0,Y 531.009,Z 376.965,A -85,B 0,C 180,E1 -4458.566,E2 -4458.566} C_VEL
LIN {X 0,Y 530.97,Z 376.971,A -85,B 0,C 180,E1 -4461.346,E2 -4461.346} C_VEL
LIN {X 0,Y 530.984,Z 376.972,A -85,B 0,C 180,E1 -4464.382,E2 -4464.382} C_VEL
LIN {X 0,Y 530.972,Z 376.97,A -85,B 0,C 180,E1 -4467.134,E2 -4467.134} C_VEL
LIN {X 0,Y 530.971,Z 376.969,A -85,B 0,C 180,E1 -4469.803,E2 -4469.803} C_VEL
LIN {X 0,Y 531.017,Z 376.968,A -85,B 0,C 180,E1 -4472.467,E2 -4472.467} C_VEL
LIN {X 0,Y 530.997,Z 376.965,A -85,B 0,C 180,E1 -4474.942,E2 -4474.942} C_VEL
LIN {X 0,Y 530.973,Z 376.968,A -85,B 0,C 180,E1 -4478.247,E2 -4478.247} C_VEL
LIN {X 0,Y 530.999,Z 376.969,A -85,B 0,C 180,E1 -4480.677,E2 -4480.677} C_VEL
LIN {X 0,Y 530.988,Z 376.966,A -85,B 0,C 180,E1 -4483.071,E2 -4483.071} C_VEL
LIN {X 0,Y 531.043,Z 376.964,A -85,B 0,C 180,E1 -4485.437,E2 -4485.437} C_VEL
LIN {X 0,Y 531.04,Z 376.964,A -85,B 0,C 180,E1 -4488.55,E2 -4488.55} C_VEL
LIN {X 0,Y 531.058,Z 376.96,A -85,B 0,C 180,E1 -4491.63,E2 -4491.63} C_VEL
LIN {X 0,Y 531.123,Z 376.95,A -85,B 0,C 180,E1 -4494.685,E2 -4494.685} C_VEL
LIN {X 0,Y 531.141,Z 376.947,A -85,B 0,C 180,E1 -4497.725,E2 -4497.725} C_VEL
LIN {X 0,Y 531.155,Z 376.945,A -85,B 0,C 180,E1 -4500.758,E2 -4500.758} C_VEL
LIN {X 0,Y 531.108,Z 376.954,A -85,B 0,C 180,E1 -4503.034,E2 -4503.034} C_VEL
LIN {X 0,Y 531.086,Z 376.955,A -85,B 0,C 180,E1 -4506.077,E2 -4506.077} C_VEL
LIN {X 0,Y 531.031,Z 376.961,A -85,B 0,C 180,E1 -4509.138,E2 -4509.138} C_VEL
LIN {X 0,Y 531.043,Z 376.959,A -85,B 0,C 180,E1 -4512.225,E2 -4512.225} C_VEL
LIN {X 0,Y 530.998,Z 376.965,A -85,B 0,C 180,E1 -4515.35,E2 -4515.35} C_VEL
LIN {X 0,Y 530.995,Z 376.965,A -85,B 0,C 180,E1 -4518.521,E2 -4518.521} C_VEL
LIN {X 0,Y 531.003,Z 376.968,A -85,B 0,C 180,E1 -4520.938,E2 -4520.938} C_VEL
LIN {X 0,Y 530.983,Z 376.971,A -85,B 0,C 180,E1 -4524.224,E2 -4524.224} C_VEL
LIN {X 0,Y 531.007,Z 376.964,A -85,B 0,C 180,E1 -4526.744,E2 -4526.744} C_VEL
LIN {X 0,Y 530.984,Z 376.971,A -85,B 0,C 180,E1 -4529.323,E2 -4529.323} C_VEL
LIN {X 0,Y 530.968,Z 376.971,A -85,B 0,C 180,E1 -4532.1,E2 -4532.1} C_VEL
LIN {X 0,Y 530.992,Z 376.966,A -85,B 0,C 180,E1 -4534.854,E2 -4534.854} C_VEL
LIN {X 0,Y 530.976,Z 376.971,A -85,B 0,C 180,E1 -4537.507,E2 -4537.507} C_VEL
LIN {X 0,Y 530.986,Z 376.971,A -85,B 0,C 180,E1 -4540.433,E2 -4540.433} C_VEL
LIN {X 0,Y 530.966,Z 376.97,A -85,B 0,C 180,E1 -4543.281,E2 -4543.281} C_VEL
LIN {X 0,Y 530.959,Z 376.972,A -85,B 0,C 180,E1 -4543.567,E2 -4543.567} C_VEL
LIN {X 0,Y 530.289,Z 377.056,A -85,B 0,C 180,E1 -4544.2,E2 -4544.2} C_VEL
LIN {X 0,Y 527.445,Z 377.412,A -85,B 0,C 180,E1 -4545.229,E2 -4545.229} C_VEL
LIN {X 0,Y 525.043,Z 377.713,A -85,B 0,C 180,E1 -4546.058,E2 -4546.058} C_VEL
LIN {X 0,Y 524.011,Z 377.84,A -85,B 0,C 180,E1 -4546.697,E2 -4546.697} C_VEL
LIN {X 0,Y 523.926,Z 377.849,A -85,B 0,C 180,E1 -4546.914,E2 -4546.914} C_VEL
LIN {X 0,Y 523.939,Z 377.848,A -85,B 0,C 180,E1 -4549.87,E2 -4549.87} C_VEL
LIN {X 0,Y 523.975,Z 378.383,A -85,B 0,C 180,E1 -4551.073,E2 -4551.073} C_VEL
LIN {X 0,Y 524.053,Z 382.442,A -85,B 0,C 180,E1 -4553.577,E2 -4553.577} C_VEL
LIN {X 0,Y 523.947,Z 387.59,A -85,B 0,C 180,E1 -4556.636,E2 -4556.636} C_VEL
LIN {X 0,Y 523.844,Z 392.301,A -85,B 0,C 180,E1 -4559.348,E2 -4559.348} C_VEL
LIN {X 0,Y 523.746,Z 397.636,A -85,B 0,C 180,E1 -4562.33,E2 -4562.33} C_VEL
LIN {X 0,Y 523.66,Z 403.309,A -85,B 0,C 180,E1 -4565.415,E2 -4565.415} C_VEL
LIN {X 0,Y 523.623,Z 407.977,A -85,B 0,C 180,E1 -4567.925,E2 -4567.925} C_VEL
LIN {X 0,Y 523.516,Z 412.654,A -85,B 0,C 180,E1 -4570.39,E2 -4570.39} C_VEL
LIN {X 0,Y 523.459,Z 418.647,A -85,B 0,C 180,E1 -4573.492,E2 -4573.492} C_VEL
LIN {X 0,Y 526.302,Z 432.013,A -85,B 0,C 180,E1 -4573.872,E2 -4573.872} C_VEL
LIN {X 0,Y 526.094,Z 445.975,A -85,B 0,C 180,E1 -4574.314,E2 -4574.314} C_VEL
LIN {X 0,Y 525.753,Z 459.311,A -85,B 0,C 180,E1 -4574.89,E2 -4574.89} C_VEL
LIN {X 0,Y 525.4,Z 471.569,A -85,B 0,C 180,E1 -4575.574,E2 -4575.574} C_VEL
LIN {X 0,Y 524.987,Z 484.182,A -85,B 0,C 180,E1 -4576.451,E2 -4576.451} C_VEL
LIN {X 0,Y 524.606,Z 495.569,A -85,B 0,C 180,E1 -4577.426,E2 -4577.426} C_VEL
LIN {X 0,Y 524.332,Z 505.006,A -85,B 0,C 180,E1 -4578.401,E2 -4578.401} C_VEL
LIN {X 0,Y 524.015,Z 514.486,A -85,B 0,C 180,E1 -4579.569,E2 -4579.569} C_VEL
LIN {X 0,Y 523.754,Z 523.545,A -85,B 0,C 180,E1 -4580.929,E2 -4580.929} C_VEL
LIN {X 0,Y 523.575,Z 530.844,A -85,B 0,C 180,E1 -4582.286,E2 -4582.286} C_VEL
LIN {X 0,Y 523.469,Z 537.402,A -85,B 0,C 180,E1 -4583.834,E2 -4583.834} C_VEL
LIN {X 0,Y 523.376,Z 541.258,A -85,B 0,C 180,E1 -4584.993,E2 -4584.993} C_VEL
LIN {X 0,Y 523.419,Z 544.216,A -85,B 0,C 180,E1 -4586.151,E2 -4586.151} C_VEL
LIN {X 0,Y 523.334,Z 546.94,A -85,B 0,C 180,E1 -4587.691,E2 -4587.691} C_VEL
LIN {X 0,Y 523.246,Z 548.309,A -85,B 0,C 180,E1 -4589.23,E2 -4589.23} C_VEL
LIN {X 0,Y 523.247,Z 548.353,A -85,B 0,C 180,E1 -4590.77,E2 -4590.77} C_VEL
LIN {X 0,Y 523.333,Z 547.066,A -85,B 0,C 180,E1 -4592.309,E2 -4592.309} C_VEL
LIN {X 0,Y 523.419,Z 544.42,A -85,B 0,C 180,E1 -4593.85,E2 -4593.85} C_VEL
LIN {X 0,Y 523.448,Z 540.345,A -85,B 0,C 180,E1 -4595.393,E2 -4595.393} C_VEL
LIN {X 0,Y 523.496,Z 534.715,A -85,B 0,C 180,E1 -4596.94,E2 -4596.94} C_VEL
LIN {X 0,Y 523.654,Z 528.359,A -85,B 0,C 180,E1 -4598.295,E2 -4598.295} C_VEL
LIN {X 0,Y 523.843,Z 520.457,A -85,B 0,C 180,E1 -4599.654,E2 -4599.654} C_VEL
LIN {X 0,Y 524.105,Z 512.203,A -85,B 0,C 180,E1 -4600.821,E2 -4600.821} C_VEL
LIN {X 0,Y 524.43,Z 502.523,A -85,B 0,C 180,E1 -4601.96,E2 -4601.96} C_VEL
LIN {X 0,Y 524.75,Z 491.206,A -85,B 0,C 180,E1 -4603.062,E2 -4603.062} C_VEL
LIN {X 0,Y 525.126,Z 480.196,A -85,B 0,C 180,E1 -4603.94,E2 -4603.94} C_VEL
LIN {X 0,Y 525.525,Z 468.252,A -85,B 0,C 180,E1 -4604.72,E2 -4604.72} C_VEL
LIN {X 0,Y 525.853,Z 455.068,A -85,B 0,C 180,E1 -4605.404,E2 -4605.404} C_VEL
LIN {X 0,Y 526.131,Z 441.026,A -85,B 0,C 180,E1 -4605.954,E2 -4605.954} C_VEL
LIN {X 0,Y 526.146,Z 431.142,A -85,B 0,C 180,E1 -4606.247,E2 -4606.247} C_VEL
LIN {X 0,Y 523.462,Z 418.661,A -85,B 0,C 180,E1 -4606.602,E2 -4606.602} C_VEL
LIN {X 0,Y 523.521,Z 412.881,A -85,B 0,C 180,E1 -4609.61,E2 -4609.61} C_VEL
LIN {X 0,Y 523.601,Z 408.024,A -85,B 0,C 180,E1 -4612.157,E2 -4612.157} C_VEL
LIN {X 0,Y 523.658,Z 403.462,A -85,B 0,C 180,E1 -4614.586,E2 -4614.586} C_VEL
LIN {X 0,Y 523.746,Z 397.798,A -85,B 0,C 180,E1 -4617.67,E2 -4617.67} C_VEL
LIN {X 0,Y 523.845,Z 392.46,A -85,B 0,C 180,E1 -4620.652,E2 -4620.652} C_VEL
LIN {X 0,Y 523.966,Z 387.111,A -85,B 0,C 180,E1 -4623.735,E2 -4623.735} C_VEL
LIN {X 0,Y 524.054,Z 382.592,A -85,B 0,C 180,E1 -4626.423,E2 -4626.423} C_VEL
LIN {X 0,Y 523.97,Z 378.289,A -85,B 0,C 180,E1 -4629.081,E2 -4629.081} C_VEL
LIN {X 0,Y 523.94,Z 377.85,A -85,B 0,C 180,E1 -4630.13,E2 -4630.13} C_VEL
LIN {X 0,Y 523.928,Z 377.851,A -85,B 0,C 180,E1 -4633.166,E2 -4633.166} C_VEL
LIN {X 0,Y 523.944,Z 377.845,A -85,B 0,C 180,E1 -4635.772,E2 -4635.772} C_VEL
LIN {X 0,Y 523.944,Z 377.845,A -85,B 0,C 180,E1 -4638.908,E2 -4638.908} C_VEL
LIN {X 0,Y 523.919,Z 377.846,A -85,B 0,C 180,E1 -4641.898,E2 -4641.898} C_VEL
LIN {X 0,Y 523.942,Z 377.845,A -85,B 0,C 180,E1 -4644.909,E2 -4644.909} C_VEL
LIN {X 0,Y 523.938,Z 377.849,A -85,B 0,C 180,E1 -4647.68,E2 -4647.68} C_VEL
LIN {X 0,Y 523.957,Z 377.845,A -85,B 0,C 180,E1 -4650.676,E2 -4650.676} C_VEL
LIN {X 0,Y 523.978,Z 377.841,A -85,B 0,C 180,E1 -4653.729,E2 -4653.729} C_VEL
LIN {X 0,Y 523.93,Z 377.845,A -85,B 0,C 180,E1 -4656.27,E2 -4656.27} C_VEL
LIN {X 0,Y 523.95,Z 377.846,A -85,B 0,C 180,E1 -4658.767,E2 -4658.767} C_VEL
LIN {X 0,Y 523.953,Z 377.843,A -85,B 0,C 180,E1 -4661.221,E2 -4661.221} C_VEL
LIN {X 0,Y 523.94,Z 377.848,A -85,B 0,C 180,E1 -4663.639,E2 -4663.639} C_VEL
LIN {X 0,Y 523.948,Z 377.843,A -85,B 0,C 180,E1 -4666.028,E2 -4666.028} C_VEL
LIN {X 0,Y 524.016,Z 377.837,A -85,B 0,C 180,E1 -4668.394,E2 -4668.394} C_VEL
LIN {X 0,Y 524.007,Z 377.836,A -85,B 0,C 180,E1 -4671.516,E2 -4671.516} C_VEL
LIN {X 0,Y 524.085,Z 377.826,A -85,B 0,C 180,E1 -4674.614,E2 -4674.614} C_VEL
LIN {X 0,Y 524.113,Z 377.822,A -85,B 0,C 180,E1 -4677.694,E2 -4677.694} C_VEL
LIN {X 0,Y 524.127,Z 377.82,A -85,B 0,C 180,E1 -4680.768,E2 -4680.768} C_VEL
LIN {X 0,Y 524.076,Z 377.831,A -85,B 0,C 180,E1 -4683.075,E2 -4683.075} C_VEL
LIN {X 0,Y 524.048,Z 377.832,A -85,B 0,C 180,E1 -4686.159,E2 -4686.159} C_VEL
LIN {X 0,Y 523.997,Z 377.838,A -85,B 0,C 180,E1 -4689.262,E2 -4689.262} C_VEL
LIN {X 0,Y 524.006,Z 377.837,A -85,B 0,C 180,E1 -4691.739,E2 -4691.739} C_VEL
LIN {X 0,Y 523.998,Z 377.838,A -85,B 0,C 180,E1 -4695.053,E2 -4695.053} C_VEL
LIN {X 0,Y 523.968,Z 377.845,A -85,B 0,C 180,E1 -4697.969,E2 -4697.969} C_VEL
LIN {X 0,Y 523.976,Z 377.84,A -85,B 0,C 180,E1 -4700.41,E2 -4700.41} C_VEL
LIN {X 0,Y 523.92,Z 377.849,A -85,B 0,C 180,E1 -4702.893,E2 -4702.893} C_VEL
LIN {X 0,Y 523.956,Z 377.842,A -85,B 0,C 180,E1 -4705.419,E2 -4705.419} C_VEL
LIN {X 0,Y 523.972,Z 377.841,A -85,B 0,C 180,E1 -4707.999,E2 -4707.999} C_VEL
LIN {X 0,Y 523.947,Z 377.849,A -85,B 0,C 180,E1 -4710.855,E2 -4710.855} C_VEL
LIN {X 0,Y 523.964,Z 377.844,A -85,B 0,C 180,E1 -4713.735,E2 -4713.735} C_VEL
LIN {X 0,Y 523.926,Z 377.847,A -85,B 0,C 180,E1 -4716.404,E2 -4716.404} C_VEL
LIN {X 0,Y 523.962,Z 377.847,A -85,B 0,C 180,E1 -4719.081,E2 -4719.081} C_VEL
LIN {X 0,Y 523.959,Z 377.848,A -85,B 0,C 180,E1 -4722.118,E2 -4722.118} C_VEL
LIN {X 0,Y 523.947,Z 377.849,A -85,B 0,C 180,E1 -4725.31,E2 -4725.31} C_VEL
LIN {X 0,Y 523.964,Z 377.847,A -85,B 0,C 180,E1 -4728.689,E2 -4728.689} C_VEL
LIN {X 0,Y 523.981,Z 377.851,A -85,B 0,C 180,E1 -4729.923,E2 -4729.923} C_VEL
LIN {X 0,Y 524.3,Z 381.556,A -85,B 0,C 180,E1 -4731.931,E2 -4731.931} C_VEL
LIN {X 0,Y 524.254,Z 385.26,A -85,B 0,C 180,E1 -4733.853,E2 -4733.853} C_VEL
LIN {X 0,Y 524.115,Z 390.832,A -85,B 0,C 180,E1 -4736.648,E2 -4736.648} C_VEL
LIN {X 0,Y 523.999,Z 396.415,A -85,B 0,C 180,E1 -4739.358,E2 -4739.358} C_VEL
LIN {X 0,Y 523.854,Z 402.666,A -85,B 0,C 180,E1 -4742.307,E2 -4742.307} C_VEL
LIN {X 0,Y 523.725,Z 409.49,A -85,B 0,C 180,E1 -4745.418,E2 -4745.418} C_VEL
LIN {X 0,Y 523.689,Z 415.108,A -85,B 0,C 180,E1 -4747.928,E2 -4747.928} C_VEL
LIN {X 0,Y 523.609,Z 420.715,A -85,B 0,C 180,E1 -4750.394,E2 -4750.394} C_VEL
LIN {X 0,Y 523.514,Z 427.794,A -85,B 0,C 180,E1 -4753.447,E2 -4753.447} C_VEL
LIN {X 0,Y 526.339,Z 441.917,A -85,B 0,C 180,E1 -4753.83,E2 -4753.83} C_VEL
LIN {X 0,Y 526.053,Z 456.152,A -85,B 0,C 180,E1 -4754.28,E2 -4754.28} C_VEL
LIN {X 0,Y 525.707,Z 470.061,A -85,B 0,C 180,E1 -4754.889,E2 -4754.889} C_VEL
LIN {X 0,Y 525.37,Z 482.153,A -85,B 0,C 180,E1 -4755.573,E2 -4755.573} C_VEL
LIN {X 0,Y 525.028,Z 493.377,A -85,B 0,C 180,E1 -4756.354,E2 -4756.354} C_VEL
LIN {X 0,Y 524.624,Z 504.92,A -85,B 0,C 180,E1 -4757.328,E2 -4757.328} C_VEL
LIN {X 0,Y 524.323,Z 515.377,A -85,B 0,C 180,E1 -4758.401,E2 -4758.401} C_VEL
LIN {X 0,Y 524.009,Z 524.821,A -85,B 0,C 180,E1 -4759.568,E2 -4759.568} C_VEL
LIN {X 0,Y 523.761,Z 533.801,A -85,B 0,C 180,E1 -4760.928,E2 -4760.928} C_VEL
LIN {X 0,Y 523.569,Z 541.054,A -85,B 0,C 180,E1 -4762.286,E2 -4762.286} C_VEL
LIN {X 0,Y 523.474,Z 547.568,A -85,B 0,C 180,E1 -4763.834,E2 -4763.834} C_VEL
LIN {X 0,Y 523.376,Z 551.38,A -85,B 0,C 180,E1 -4764.993,E2 -4764.993} C_VEL
LIN {X 0,Y 523.419,Z 554.316,A -85,B 0,C 180,E1 -4766.15,E2 -4766.15} C_VEL
LIN {X 0,Y 523.333,Z 557.002,A -85,B 0,C 180,E1 -4767.691,E2 -4767.691} C_VEL
LIN {X 0,Y 523.247,Z 558.334,A -85,B 0,C 180,E1 -4769.23,E2 -4769.23} C_VEL
LIN {X 0,Y 523.247,Z 558.334,A -85,B 0,C 180,E1 -4770.77,E2 -4770.77} C_VEL
LIN {X 0,Y 523.333,Z 557.005,A -85,B 0,C 180,E1 -4772.309,E2 -4772.309} C_VEL
LIN {X 0,Y 523.419,Z 554.32,A -85,B 0,C 180,E1 -4773.849,E2 -4773.849} C_VEL
LIN {X 0,Y 523.452,Z 550.201,A -85,B 0,C 180,E1 -4775.393,E2 -4775.393} C_VEL
LIN {X 0,Y 523.495,Z 544.526,A -85,B 0,C 180,E1 -4776.94,E2 -4776.94} C_VEL
LIN {X 0,Y 523.664,Z 538.127,A -85,B 0,C 180,E1 -4778.295,E2 -4778.295} C_VEL
LIN {X 0,Y 523.863,Z 530.174,A -85,B 0,C 180,E1 -4779.654,E2 -4779.654} C_VEL
LIN {X 0,Y 524.117,Z 521.85,A -85,B 0,C 180,E1 -4780.82,E2 -4780.82} C_VEL
LIN {X 0,Y 524.449,Z 511.069,A -85,B 0,C 180,E1 -4782.068,E2 -4782.068} C_VEL
LIN {X 0,Y 524.748,Z 500.612,A -85,B 0,C 180,E1 -4783.062,E2 -4783.062} C_VEL
LIN {X 0,Y 525.191,Z 488.046,A -85,B 0,C 180,E1 -4784.037,E2 -4784.037} C_VEL
LIN {X 0,Y 525.587,Z 475.57,A -85,B 0,C 180,E1 -4784.817,E2 -4784.817} C_VEL
LIN {X 0,Y 525.887,Z 462.744,A -85,B 0,C 180,E1 -4785.453,E2 -4785.453} C_VEL
LIN {X 0,Y 526.205,Z 448.767,A -85,B 0,C 180,E1 -4785.974,E2 -4785.974} C_VEL
LIN {X 0,Y 526.228,Z 440.584,A -85,B 0,C 180,E1 -4786.209,E2 -4786.209} C_VEL
LIN {X 0,Y 523.512,Z 427.678,A -85,B 0,C 180,E1 -4786.575,E2 -4786.575} C_VEL
LIN {X 0,Y 523.607,Z 420.631,A -85,B 0,C 180,E1 -4789.606,E2 -4789.606} C_VEL
LIN {X 0,Y 523.68,Z 414.788,A -85,B 0,C 180,E1 -4792.179,E2 -4792.179} C_VEL
LIN {X 0,Y 523.72,Z 409.446,A -85,B 0,C 180,E1 -4794.582,E2 -4794.582} C_VEL
LIN {X 0,Y 523.852,Z 402.665,A -85,B 0,C 180,E1 -4797.692,E2 -4797.692} C_VEL
LIN {X 0,Y 523.998,Z 396.414,A -85,B 0,C 180,E1 -4800.642,E2 -4800.642} C_VEL
LIN {X 0,Y 524.137,Z 389.995,A -85,B 0,C 180,E1 -4803.763,E2 -4803.763} C_VEL
LIN {X 0,Y 524.28,Z 384.649,A -85,B 0,C 180,E1 -4806.457,E2 -4806.457} C_VEL
LIN {X 0,Y 524.229,Z 379.697,A -85,B 0,C 180,E1 -4809.057,E2 -4809.057} C_VEL
LIN {X 0,Y 523.996,Z 377.845,A -85,B 0,C 180,E1 -4810.137,E2 -4810.137} C_VEL
LIN {X 0,Y 523.923,Z 377.851,A -85,B 0,C 180,E1 -4813.167,E2 -4813.167} C_VEL
LIN {X 0,Y 523.932,Z 377.848,A -85,B 0,C 180,E1 -4815.771,E2 -4815.771} C_VEL
LIN {X 0,Y 523.963,Z 377.843,A -85,B 0,C 180,E1 -4818.91,E2 -4818.91} C_VEL
LIN {X 0,Y 523.921,Z 377.847,A -85,B 0,C 180,E1 -4821.899,E2 -4821.899} C_VEL
LIN {X 0,Y 523.94,Z 377.845,A -85,B 0,C 180,E1 -4824.909,E2 -4824.909} C_VEL
LIN {X 0,Y 523.939,Z 377.849,A -85,B 0,C 180,E1 -4827.679,E2 -4827.679} C_VEL
LIN {X 0,Y 523.956,Z 377.847,A -85,B 0,C 180,E1 -4830.676,E2 -4830.676} C_VEL
LIN {X 0,Y 523.976,Z 377.842,A -85,B 0,C 180,E1 -4833.729,E2 -4833.729} C_VEL
LIN {X 0,Y 523.927,Z 377.846,A -85,B 0,C 180,E1 -4836.27,E2 -4836.27} C_VEL
LIN {X 0,Y 523.948,Z 377.847,A -85,B 0,C 180,E1 -4838.767,E2 -4838.767} C_VEL
LIN {X 0,Y 523.955,Z 377.842,A -85,B 0,C 180,E1 -4841.221,E2 -4841.221} C_VEL
LIN {X 0,Y 523.939,Z 377.848,A -85,B 0,C 180,E1 -4843.639,E2 -4843.639} C_VEL
LIN {X 0,Y 523.948,Z 377.843,A -85,B 0,C 180,E1 -4846.028,E2 -4846.028} C_VEL
LIN {X 0,Y 524.015,Z 377.837,A -85,B 0,C 180,E1 -4848.394,E2 -4848.394} C_VEL
LIN {X 0,Y 524.006,Z 377.837,A -85,B 0,C 180,E1 -4851.516,E2 -4851.516} C_VEL
LIN {X 0,Y 524.085,Z 377.826,A -85,B 0,C 180,E1 -4854.614,E2 -4854.614} C_VEL
LIN {X 0,Y 524.113,Z 377.822,A -85,B 0,C 180,E1 -4857.695,E2 -4857.695} C_VEL
LIN {X 0,Y 524.125,Z 377.821,A -85,B 0,C 180,E1 -4860.768,E2 -4860.768} C_VEL
LIN {X 0,Y 524.074,Z 377.831,A -85,B 0,C 180,E1 -4863.075,E2 -4863.075} C_VEL
LIN {X 0,Y 524.048,Z 377.833,A -85,B 0,C 180,E1 -4866.159,E2 -4866.159} C_VEL
LIN {X 0,Y 523.999,Z 377.837,A -85,B 0,C 180,E1 -4869.262,E2 -4869.262} C_VEL
LIN {X 0,Y 524.005,Z 377.837,A -85,B 0,C 180,E1 -4871.739,E2 -4871.739} C_VEL
LIN {X 0,Y 523.997,Z 377.838,A -85,B 0,C 180,E1 -4875.053,E2 -4875.053} C_VEL
LIN {X 0,Y 523.967,Z 377.845,A -85,B 0,C 180,E1 -4877.969,E2 -4877.969} C_VEL
LIN {X 0,Y 523.975,Z 377.84,A -85,B 0,C 180,E1 -4880.41,E2 -4880.41} C_VEL
LIN {X 0,Y 523.92,Z 377.85,A -85,B 0,C 180,E1 -4882.893,E2 -4882.893} C_VEL
LIN {X 0,Y 523.955,Z 377.843,A -85,B 0,C 180,E1 -4885.419,E2 -4885.419} C_VEL
LIN {X 0,Y 523.972,Z 377.841,A -85,B 0,C 180,E1 -4887.999,E2 -4887.999} C_VEL
LIN {X 0,Y 523.947,Z 377.849,A -85,B 0,C 180,E1 -4890.855,E2 -4890.855} C_VEL
LIN {X 0,Y 523.964,Z 377.843,A -85,B 0,C 180,E1 -4893.735,E2 -4893.735} C_VEL
LIN {X 0,Y 523.926,Z 377.846,A -85,B 0,C 180,E1 -4896.404,E2 -4896.404} C_VEL
LIN {X 0,Y 523.925,Z 377.85,A -85,B 0,C 180,E1 -4899.085,E2 -4899.085} C_VEL
LIN {X 0,Y 523.958,Z 377.847,A -85,B 0,C 180,E1 -4902.119,E2 -4902.119} C_VEL
LIN {X 0,Y 523.958,Z 377.847,A -85,B 0,C 180,E1 -4905.309,E2 -4905.309} C_VEL
LIN {X 0,Y 523.926,Z 377.849,A -85,B 0,C 180,E1 -4906.914,E2 -4906.914} C_VEL
LIN {X 0,Y 523.253,Z 377.949,A -85,B 0,C 180,E1 -4907.555,E2 -4907.555} C_VEL
LIN {X 0,Y 520.389,Z 378.292,A -85,B 0,C 180,E1 -4908.597,E2 -4908.597} C_VEL
LIN {X 0,Y 517.977,Z 378.589,A -85,B 0,C 180,E1 -4909.436,E2 -4909.436} C_VEL
LIN {X 0,Y 516.948,Z 378.721,A -85,B 0,C 180,E1 -4910.084,E2 -4910.084} C_VEL
LIN {X 0,Y 516.869,Z 378.743,A -85,B 0,C 180,E1 -4910.303,E2 -4910.303} C_VEL
LIN {X 0,Y 516.893,Z 378.986,A -85,B 0,C 180,E1 -4910.806,E2 -4910.806} C_VEL
LIN {X 0,Y 517.023,Z 383.001,A -85,B 0,C 180,E1 -4913.322,E2 -4913.322} C_VEL
LIN {X 0,Y 516.932,Z 387.622,A -85,B 0,C 180,E1 -4916.122,E2 -4916.122} C_VEL
LIN {X 0,Y 516.835,Z 392.443,A -85,B 0,C 180,E1 -4918.947,E2 -4918.947} C_VEL
LIN {X 0,Y 516.699,Z 397.063,A -85,B 0,C 180,E1 -4921.572,E2 -4921.572} C_VEL
LIN {X 0,Y 516.635,Z 401.774,A -85,B 0,C 180,E1 -4924.195,E2 -4924.195} C_VEL
LIN {X 0,Y 516.54,Z 406.495,A -85,B 0,C 180,E1 -4926.761,E2 -4926.761} C_VEL
LIN {X 0,Y 516.475,Z 412.278,A -85,B 0,C 180,E1 -4929.872,E2 -4929.872} C_VEL
LIN {X 0,Y 516.398,Z 418.732,A -85,B 0,C 180,E1 -4933.266,E2 -4933.266} C_VEL
LIN {X 0,Y 519.493,Z 433.01,A -85,B 0,C 180,E1 -4933.679,E2 -4933.679} C_VEL
LIN {X 0,Y 519.256,Z 446.646,A -85,B 0,C 180,E1 -4934.124,E2 -4934.124} C_VEL
LIN {X 0,Y 518.899,Z 459.392,A -85,B 0,C 180,E1 -4934.686,E2 -4934.686} C_VEL
LIN {X 0,Y 518.524,Z 471.648,A -85,B 0,C 180,E1 -4935.378,E2 -4935.378} C_VEL
LIN {X 0,Y 518.133,Z 482.97,A -85,B 0,C 180,E1 -4936.169,E2 -4936.169} C_VEL
LIN {X 0,Y 517.697,Z 494.577,A -85,B 0,C 180,E1 -4937.156,E2 -4937.156} C_VEL
LIN {X 0,Y 517.339,Z 505.081,A -85,B 0,C 180,E1 -4938.242,E2 -4938.242} C_VEL
LIN {X 0,Y 517.013,Z 514.56,A -85,B 0,C 180,E1 -4939.426,E2 -4939.426} C_VEL
LIN {X 0,Y 516.726,Z 523.606,A -85,B 0,C 180,E1 -4940.804,E2 -4940.804} C_VEL
LIN {X 0,Y 516.508,Z 530.888,A -85,B 0,C 180,E1 -4942.18,E2 -4942.18} C_VEL
LIN {X 0,Y 516.386,Z 537.43,A -85,B 0,C 180,E1 -4943.749,E2 -4943.749} C_VEL
LIN {X 0,Y 516.305,Z 541.275,A -85,B 0,C 180,E1 -4944.924,E2 -4944.924} C_VEL
LIN {X 0,Y 516.325,Z 544.225,A -85,B 0,C 180,E1 -4946.098,E2 -4946.098} C_VEL
LIN {X 0,Y 516.26,Z 546.942,A -85,B 0,C 180,E1 -4947.659,E2 -4947.659} C_VEL
LIN {X 0,Y 516.156,Z 548.309,A -85,B 0,C 180,E1 -4949.22,E2 -4949.22} C_VEL
LIN {X 0,Y 516.157,Z 548.352,A -85,B 0,C 180,E1 -4950.78,E2 -4950.78} C_VEL
LIN {X 0,Y 516.26,Z 547.066,A -85,B 0,C 180,E1 -4952.341,E2 -4952.341} C_VEL
LIN {X 0,Y 516.325,Z 544.425,A -85,B 0,C 180,E1 -4953.903,E2 -4953.903} C_VEL
LIN {X 0,Y 516.381,Z 540.36,A -85,B 0,C 180,E1 -4955.467,E2 -4955.467} C_VEL
LIN {X 0,Y 516.408,Z 534.744,A -85,B 0,C 180,E1 -4957.036,E2 -4957.036} C_VEL
LIN {X 0,Y 516.592,Z 528.402,A -85,B 0,C 180,E1 -4958.41,E2 -4958.41} C_VEL
